METHOD PRIVATE ActionRun
VAR_INPUT
	tempActStep:ITFActStep;
END_VAR
VAR
END_VAR
VAR_STAT//此处定义静态变量, 保证每次进入该函数时能够在线监控当前值
	tempStep:DINT;
END_VAR
tempStep:=tempActStep.getStep();
CASE tempStep OF
0:
	IF tempActStep.isEx() THEN
		tempActStep.setBusyFlag();
		tempActStep.toBeginStep();
	END_IF
	t1(IN:= FALSE );
	t2(IN:= FALSE );
	t3(IN:= FALSE );
10:
	gShowLogTextTitle:='Chamber LL Vent';
	IF gRunningState<>RunningStatus.eErrorState THEN
		tempActStep.addStep(10,FALSE);
	ELSE
		gRunningLog.append(CONCAT('Chamber Vent POU Run:',DINT_TO_STRING(tempStep)));
		gRunningLog.append('Chamber Vent POU Run: Running State Error');
		error_Trigger(105);
		tempActStep.toDoneStep();
	END_IF
20:
	IF NOT gICP.ForeLineGauge.error AND gICP.ForeLineGauge.outputValue<gRoughtPumVaccum*10 THEN
		tempActStep.addStep(10,FALSE);
	ELSE
		error_Trigger(107);
		tempActStep.toDoneStep();
	END_IF
30:
	tempActStep.toStep(100,FALSE);
	gRoughRemain:=FALSE;
100:
	tempActStep.addStep(10,TRUE);
110:
	S_RoughPumping.Act_Init_Status();
	S_RoughPumping.Act_Ex();
	tempActStep.addStep(10,FALSE);
120:
	IF S_RoughPumping.done THEN
		tempActStep.addStep(2,FALSE);
	END_IF
	IF S_RoughPumping.errDone THEN
		tempActStep.toErrDoneStep();
	END_IF
122:
	tempActStep.addStep(2,TRUE);
124:
	IF gICP.TruboPum.Act_Close() THEN
		gRunningLog.append(CONCAT('Chamber Vent POU Run:',DINT_TO_STRING(tempStep)));
		gRunningLog.append('Chamber Vent POU Run: TruboPum Close');
		tempActStep.addStep(2,FALSE);
	END_IF
126:
	IF (gICP.TruboPum.Get_Done_Close() AND gICP.TruboPumNoRotation) AND 
		(NOT gICP.TruboPumAcc AND NOT gICP.TruboPumDcc AND NOT gICP.TruboPumNormal AND gICP.TruboPumNoRotation) THEN
		gRunningLog.append(CONCAT('Chamber Vent POU Run:',DINT_TO_STRING(tempStep)));
		gRunningLog.append('Chamber Vent POU Run: TruboPum Close Done');
		tempActStep.addStep(2,FALSE);
	END_IF
128:
	tempActStep.addStep(2,FALSE);
130:
	tempActStep.addStep(10,TRUE);
140:
	IF gICP.GateDoorValve.Get_Done_Ret() AND gICP.GateDoorRetSensor AND
		gICP.VentValve.Get_Done_Ret() AND NOT gICP.VentExtRelay AND
		gICP.SlowPummingValve.Get_Done_Ret() AND NOT gICP.SlowPummingExtRelay AND
		gICP.FastPummingValve.Get_Done_Ret() AND NOT gICP.FastPummingExtRelay AND
		gICP.ForlinLineValve.Get_Done_Ext() AND gICP.ForlinLineValveExtRelay AND////////////////
		gICP.RoughValve.Get_Done_Ret() AND NOT gICP.RoughValveExtRelay AND
		(gICP.PDV.Get_Done_Ext() OR gICP.PDVOpenSensor) AND gICP.PDVOpenSensor  THEN///////////////
		gRunningLog.append(CONCAT('Chamber Vent POU Run:',DINT_TO_STRING(tempStep)));
		gRunningLog.append('Chamber Vent POU Run: All Main Actuator Recovery');
		tempActStep.addStep(5,FALSE);		
	END_IF
145:
	IF gICP.PDV.Act_Retract() THEN
		gRunningLog.append(CONCAT('Chamber Vent POU Run:',DINT_TO_STRING(tempStep)));
		gRunningLog.append('Chamber Vent POU Run: PDV Close');
		tempActStep.addStep(2,FALSE);	
	END_IF
147:
	IF (gICP.PDV.Get_Done_Ret() OR gICP.PDVCloseSensor) THEN
		gRunningLog.append(CONCAT('Chamber Vent POU Run:',DINT_TO_STRING(tempStep)));
		gRunningLog.append('Chamber Vent POU Run: PDV Close DOne');
		tempActStep.addStep(3,FALSE);	
	END_IF
150:
	IF gICP.GateDoorValve.Act_Extend() THEN
		gRunningLog.append(CONCAT('Chamber Vent POU Run:',DINT_TO_STRING(tempStep)));
		gRunningLog.append('Chamber Vent POU Run: Gate Door Open');
		tempActStep.addStep(10,FALSE);	
	END_IF
160:
	IF gICP.GateDoorValve.Get_Done_Ext() AND gICP.GateDoorExtSensor THEN
		gRunningLog.append(CONCAT('Chamber Vent POU Run:',DINT_TO_STRING(tempStep)));
		gRunningLog.append('Chamber Vent POU Run: Gate Door Open Done');
		tempActStep.addStep(10,FALSE);	
	END_IF
170:
	tempActStep.addStep(10,TRUE);
180:
	tempActStep.toStep(220,FALSE);	
220:
	IF gICP.VentValve.Act_Extend() THEN
		gRunningLog.append(CONCAT('Chamber Vent POU Run:',DINT_TO_STRING(tempStep)));
		gRunningLog.append('Chamber Vent POU Run: Vent Valve Open');
		gRoughRemain:=FALSE;
		gRoughRemainTMPCanOpen:=FALSE;
		ups_CX51X0.Act_Wrtie();
		tempActStep.addStep(10,FALSE);
	END_IF
230:
	IF gICP.VentValve.Get_Done_Ext() THEN
		gRunningLog.append(CONCAT('Chamber Vent POU Run:',DINT_TO_STRING(tempStep)));
		gRunningLog.append('Chamber Vent POU Run: Vent Valve Open Done');
		tempActStep.addStep(10,FALSE);
	END_IF
240:
	t2(IN:= gICP.LoadLockGauge.outputValue>gATMPressure,PT:=T#120S );
	IF t2.Q OR NOT gICP.I_LLSwitch THEN
		t1(IN:= FALSE );
		t2(IN:= FALSE );
		t3(IN:= FALSE );
		gRunningLog.append(CONCAT('Chamber Vent POU Run:',DINT_TO_STRING(tempStep)));
		gRunningLog.append(CONCAT('Chamber Vent POU Run:LL Vent Pressure Arrive：',REAL_TO_STRING(gICP.LoadLockGauge.outputValue)));
		tempActStep.addStep(10,FALSE);
		RETURN;
	END_IF
	t1(IN:= TRUE,PT:=timeOutTime );
	IF t1.Q THEN
		t1(IN:= FALSE );
		t2(IN:= FALSE );
		t3(IN:= FALSE );
		error_Trigger(108);
//		tempActStep.toStep(170,FALSE);
		tempActStep.toDoneStep();
		RETURN;
	END_IF
250:
	tempActStep.addStep(10,TRUE);
260:
	IF gICP.VentValve.Act_Retract() THEN
		gRunningLog.append(CONCAT('Chamber Vent POU Run:',DINT_TO_STRING(tempStep)));
		gRunningLog.append('Chamber Vent POU Run: Vent Valve Close');
		tempActStep.addStep(10,FALSE);
	END_IF
270:
	IF gICP.VentValve.Get_Done_Ret() THEN
		gRunningLog.append(CONCAT('Chamber Vent POU Run:',DINT_TO_STRING(tempStep)));
		gRunningLog.append('Chamber Vent POU Run: Vent Valve Close Done');
		tempActStep.addStep(10,FALSE);
	END_IF
280:
	t3(IN:=TRUE,PT:=T#1S);
	IF t3.Q THEN
		t1(IN:= FALSE );
		t2(IN:= FALSE );
		t3(IN:= FALSE );
		tempActStep.addStep(10,FALSE);
	END_IF
290:
	tempActStep.addStep(10,TRUE);
300:
	IF gICP.GateDoorValve.Act_Retract() THEN
		gRunningLog.append(CONCAT('Chamber Vent POU Run:',DINT_TO_STRING(tempStep)));
		gRunningLog.append('Chamber Vent POU Run: Gate Door Close');
		tempActStep.addStep(10,FALSE);
	END_IF
310:
	IF gICP.GateDoorValve.Get_Done_Ret() THEN
		gRunningLog.append(CONCAT('Chamber Vent POU Run:',DINT_TO_STRING(tempStep)));
		gRunningLog.append('Chamber Vent POU Run: Gate Door Close Done');
		tempActStep.addStep(10,FALSE);
	END_IF
320:
	tempActStep.toStep(370,FALSE);
370:
	tempActStep.addStep(10,TRUE);
380:
	IF gICP.ForlinLineValve.Act_Extend() THEN
		gRunningLog.append(CONCAT('Chamber Vent POU Run:',DINT_TO_STRING(tempStep)));
		gRunningLog.append('Chamber Vent POU Run: ForLine Valve Open');
		tempActStep.addStep(10,FALSE);
	END_IF
390:
	IF gICP.ForlinLineValve.Get_Done_Ext() THEN
		gRunningLog.append(CONCAT('Chamber Vent POU Run:',DINT_TO_STRING(tempStep)));
		gRunningLog.append('Chamber Vent POU Run: ForLine Valve Open Done');
		tempActStep.addStep(10,FALSE);
	END_IF
400:
	tempActStep.toStep(1000,FALSE);
1000:
	tempActStep.toDoneStep();

60000://Done
	tempActStep.setDoneFlag();
	tempActStep.toZeroStep();
	
65000://Error
	tempActStep.setErrDoneFlag();
	tempActStep.toZeroStep();
	gICP.VentValve.Act_Retract();
END_CASE
END_METHOD

END_PROGRAM

// ---- POUs/MachinePOU/SemiAutomatic/S_MachineVent.TcPOU
PROGRAM S_MachineVent
VAR_INPUT
	bInit				:BOOL:=FALSE;// 初始化状态 busy/done/errDone
	bTrig				:BOOL:=FALSE;// 执行触发 信号
	bReset				:BOOL:=FALSE;// 报错 复位
	bPause				:BOOL:=FALSE;// 暂停 运行
	bStop				:BOOL:=FALSE;// 停止 运行
	bAbort				:BOOL:=FALSE;// 中止 运行
	
END_VAR
VAR_OUTPUT
	busy				:BOOL;
	done				:BOOL;
	errDone				:BOOL;
END_VAR
VAR
	actStep				:ActStepBase;
END_VAR
VAR
	i: INT;
	t1:ton;
	t2:ton;
	t3:ton;
	notchoose:BOOL;
	timeOutTime:TIME:=T#120S;
	safecheckTime:TIME:=T#1S;
END_VAR

busy:=actStep.isBusy();
done:=actStep.isDone();
errDone:=actStep.isError();
actStep.Act_Pause(pause:=bPause);

IF bTrig THEN
	bTrig:=FALSE;
	IF NOT busy THEN
		actStep.Act_ex();
	END_IF
END_IF

//状态复位
IF bInit THEN
	bInit:=FALSE;
	Act_init_status();
END_IF

IF bAbort OR bStop THEN
	bAbort:=FALSE;
	bStop:=FALSE;
	Act_init_status();
	actStep.toZeroStep();
	gShowLogTextTitle:='NON';
END_IF
ActionRun(tempActStep:=actStep);

(*
---Trigger action
*)
METHOD Act_Ex : BOOL
VAR_INPUT
END_VAR
IF NOT busy THEN
	actStep.Act_ex();
	Act_Ex:=TRUE;
ELSE
	Act_Ex:=FALSE;
END_IF
END_METHOD

(*
---功能: 状态复位 busy/done/errDone;
*)
METHOD Act_Init_Status
VAR_INPUT
END_VAR
actStep.Act_Init();
END_METHOD

METHOD PRIVATE ActionRun
VAR_INPUT
	tempActStep:ITFActStep;
END_VAR
VAR
END_VAR
VAR_STAT//此处定义静态变量, 保证每次进入该函数时能够在线监控当前值
	tempStep:DINT;
END_VAR
tempStep:=tempActStep.getStep();
CASE tempStep OF
0:
	IF tempActStep.isEx() THEN
		tempActStep.setBusyFlag();
		tempActStep.toBeginStep();
	END_IF
	t1(IN:= FALSE );
	t2(IN:= FALSE );
	t3(IN:= FALSE );
10:
	gShowLogTextTitle:='Machine Vent';
	IF gRunningState<>RunningStatus.eErrorState THEN
		tempActStep.addStep(10,FALSE);
	ELSE
		error_Trigger(105);
		tempActStep.toErrDoneStep();
	END_IF
20:
	IF NOT gICP.ForeLineGauge.error AND gICP.ForeLineGauge.outputValue<gRoughtPumVaccum*10 THEN
		tempActStep.addStep(10,FALSE);
	ELSE
		error_Trigger(107);
		tempActStep.toErrDoneStep();
	END_IF
30:
	gRoughRemain:=FALSE;
	tempActStep.toStep(100,FALSE);
100:
	tempActStep.addStep(10,TRUE);
110:
	S_RoughPumping.Act_Init_Status();
	S_RoughPumping.Act_Ex();
	tempActStep.addStep(10,FALSE);
120:
	IF S_RoughPumping.done THEN
		gShowLogTextTitle:='Machine Vent';
		tempActStep.addStep(10,FALSE);
	END_IF
	IF S_RoughPumping.errDone THEN
		tempActStep.toErrDoneStep();
	END_IF
130:
	tempActStep.addStep(10,TRUE);
140:
	IF gICP.TruboPum.Act_Close() THEN
		gRunningLog.append(CONCAT('Machine Vent POU Run:',DINT_TO_STRING(tempStep)));
		gRunningLog.append('Machine Vent POU Run:TB Close');
		tempActStep.addStep(10,FALSE);
	END_IF
150:
	IF (gICP.TruboPum.Get_Done_Close() AND gICP.TruboPumNoRotation) AND (NOT gICP.TruboPumAcc AND NOT gICP.TruboPumDcc AND NOT gICP.TruboPumNormal AND gICP.TruboPumNoRotation) THEN
		gRunningLog.append(CONCAT('Machine Vent POU Run:',DINT_TO_STRING(tempStep)));
		gRunningLog.append('Machine Vent POU Run:TB Close Done');
		tempActStep.addStep(10,FALSE);
	END_IF
160:
	IF gICP.GateDoorValve.Get_Done_Ret() AND gICP.GateDoorRetSensor AND
		gICP.VentValve.Get_Done_Ret() AND NOT gICP.VentExtRelay AND
		gICP.SlowPummingValve.Get_Done_Ret() AND NOT gICP.SlowPummingExtRelay AND
		gICP.FastPummingValve.Get_Done_Ret() AND NOT gICP.FastPummingExtRelay AND
		gICP.ForlinLineValve.Get_Done_Ext() AND gICP.ForlinLineValveExtRelay AND
		gICP.RoughValve.Get_Done_Ret() AND NOT gICP.RoughValveExtRelay AND
		(gICP.PDV.Get_Done_Ext() OR gICP.PDVOpenSensor)  THEN
		gRunningLog.append(CONCAT('Machine Vent POU Run:',DINT_TO_STRING(tempStep)));
		gRunningLog.append('Machine Vent POU Run:Main Actuator Recovery');
		tempActStep.addStep(10,FALSE);		
	END_IF
170:
	IF gICP.GateDoorValve.Act_Extend() THEN
		gRunningLog.append(CONCAT('Machine Vent POU Run:',DINT_TO_STRING(tempStep)));
		gRunningLog.append('Machine Vent POU Run:Gate Door Open');
		tempActStep.addStep(10,FALSE);	
	END_IF
180:
	IF gICP.GateDoorValve.Get_Done_Ext() AND gICP.GateDoorExtSensor THEN
		gRunningLog.append(CONCAT('Machine Vent POU Run:',DINT_TO_STRING(tempStep)));
		gRunningLog.append('Machine Vent POU Run:Gate Door Open Done');
		tempActStep.addStep(10,FALSE);	
	END_IF
190:
	tempActStep.addStep(10,TRUE);
200:
	tempActStep.addStep(10,FALSE);
210:
	IF gICP.PDV.Act_Open() THEN
		gRunningLog.append(CONCAT('Machine Vent POU Run:',DINT_TO_STRING(tempStep)));
		gRunningLog.append('Machine Vent POU Run:PDV Open');
		tempActStep.addStep(2,FALSE);
	END_IF
212:
	IF (gICP.PDV.Get_Done_Ext() OR gICP.PDVOpenSensor) THEN
		gRunningLog.append(CONCAT('Machine Vent POU Run:',DINT_TO_STRING(tempStep)));
		gRunningLog.append('Machine Vent POU Run:PDV Open Done');
		tempActStep.addStep(2,FALSE);
	END_IF
214:
	tempActStep.addStep(2,TRUE);
216:
	IF gICP.ForlinLineValve.Act_Retract() THEN
		gRunningLog.append(CONCAT('Machine Vent POU Run:',DINT_TO_STRING(tempStep)));
		gRunningLog.append('Machine Vent POU Run:ForeLine Valve Close');
		tempActStep.addStep(2,FALSE);
	END_IF
218:
	IF gICP.ForlinLineValve.Get_Done_Ret() THEN
		gRunningLog.append(CONCAT('Machine Vent POU Run:',DINT_TO_STRING(tempStep)));
		gRunningLog.append('Machine Vent POU Run:ForeLine Valve Close Done');
		tempActStep.addStep(2,FALSE);
	END_IF
220:
	IF gICP.VentValve.Act_Extend() THEN
		gRunningLog.append(CONCAT('Machine Vent POU Run:',DINT_TO_STRING(tempStep)));
		gRunningLog.append('Machine Vent POU Run:Vent Valve Open');
		gRoughRemain:=FALSE;
		gRoughRemainTMPCanOpen:=FALSE;
		ups_CX51X0.Act_Wrtie();
		tempActStep.addStep(10,FALSE);
	END_IF
230:
	IF gICP.VentValve.Get_Done_Ext() THEN
		gRunningLog.append(CONCAT('Machine Vent POU Run:',DINT_TO_STRING(tempStep)));
		gRunningLog.append('Machine Vent POU Run:Vent Valve Open Done');
		tempActStep.addStep(10,FALSE);
	END_IF
240:
	t2(IN:= gICP.LoadLockGauge.outputValue>gATMPressure,PT:=T#180S );
	IF t2.Q OR NOT gICP.I_LLSwitch THEN
		t1(IN:= FALSE );
		t2(IN:= FALSE );
		t3(IN:= FALSE );
		gRunningLog.append(CONCAT('Machine Vent POU Run:',DINT_TO_STRING(tempStep)));
		gRunningLog.append(CONCAT('Machine Vent POU Run:LL Vent Pressure Arrive：',REAL_TO_STRING(gICP.LoadLockGauge.outputValue)));
		tempActStep.addStep(10,FALSE);
		RETURN;
	END_IF
	t1(IN:= TRUE,PT:=timeOutTime );
	IF t1.Q THEN
		t1(IN:= FALSE );
		t2(IN:= FALSE );
		t3(IN:= FALSE );
		error_Trigger(112);
//		tempActStep.toStep(214,FALSE);
		tempActStep.toDoneStep();
		RETURN;
	END_IF
250:
	tempActStep.addStep(10,TRUE);
260:
	IF gICP.VentValve.Act_Retract() THEN
		gRunningLog.append(CONCAT('Machine Vent POU Run:',DINT_TO_STRING(tempStep)));
		gRunningLog.append('Machine Vent POU Run:Vent Valve Close');
		tempActStep.addStep(10,FALSE);
	END_IF
270:
	IF gICP.VentValve.Get_Done_Ret() THEN
		gRunningLog.append(CONCAT('Machine Vent POU Run:',DINT_TO_STRING(tempStep)));
		gRunningLog.append('Machine Vent POU Run:Vent Valve Close Done');
		tempActStep.addStep(10,FALSE);
	END_IF
280:
	t3(IN:=TRUE,PT:=T#1S);
	IF t3.Q THEN
		t1(IN:= FALSE );
		t2(IN:= FALSE );
		t3(IN:= FALSE );
		tempActStep.addStep(10,FALSE);
	END_IF
290:
	tempActStep.addStep(10,TRUE);
300:
	IF gICP.GateDoorValve.Act_Retract() THEN
		gRunningLog.append(CONCAT('Machine Vent POU Run:',DINT_TO_STRING(tempStep)));
		gRunningLog.append('Machine Vent POU Run:Gate Door Close');
		tempActStep.addStep(10,FALSE);
	END_IF
310:
	IF gICP.GateDoorValve.Get_Done_Ret() THEN
		gRunningLog.append(CONCAT('Machine Vent POU Run:',DINT_TO_STRING(tempStep)));
		gRunningLog.append('Machine Vent POU Run:Gate Door Close Done');
		tempActStep.addStep(10,FALSE);
	END_IF
320:
	tempActStep.toStep(370,FALSE);
370:
	tempActStep.addStep(10,TRUE);
380:
	IF gICP.PDV.Act_Retract() THEN
		gRunningLog.append(CONCAT('Machine Vent POU Run:',DINT_TO_STRING(tempStep)));
		gRunningLog.append('Machine Vent POU Run:PDV Close');
		tempActStep.addStep(10,FALSE);
	END_IF
390:
	IF (gICP.PDV.Get_Done_Ret() OR gICP.PDVCloseSensor) THEN
		gRunningLog.append(CONCAT('Machine Vent POU Run:',DINT_TO_STRING(tempStep)));
		gRunningLog.append('Machine Vent POU Run:PDV Close Done');
		tempActStep.addStep(10,FALSE);
	END_IF
400:
	tempActStep.toStep(1000,FALSE);
1000:
	tempActStep.toDoneStep();

60000://Done
	tempActStep.setDoneFlag();
	tempActStep.toZeroStep();
	
65000://Error
	tempActStep.setErrDoneFlag();
	tempActStep.toZeroStep();
	gICP.VentValve.Act_Retract();
END_CASE
END_METHOD

END_PROGRAM

// ---- POUs/MachinePOU/SemiAutomatic/S_Etching.TcPOU
PROGRAM S_Etching
VAR_INPUT
	bInit				:BOOL:=FALSE;// 初始化状态 busy/done/errDone
	bTrig				:BOOL:=FALSE;// 执行触发 信号
	bReset				:BOOL:=FALSE;// 报错 复位
	bPause				:BOOL:=FALSE;// 暂停 运行
	bStop				:BOOL:=FALSE;// 停止 运行
	bAbort				:BOOL:=FALSE;// 中止 运行
	
END_VAR
VAR_OUTPUT
	busy				:BOOL;
	done				:BOOL;
	errDone				:BOOL;
END_VAR
VAR
	actStep				:ActStepBase;
END_VAR
VAR
	i: INT;
	t1:ton;
	t2:ton;
	t3:ton;
	notchoose:BOOL;
	timeOutTime:TIME:= T#120S;
	ventTime:TIME:=T#15S;
	safecheckTime:TIME:=T#2S;
	currentTimes:INT:=1;
	rfComControl:TON;
	rTrig:R_TRIG;
END_VAR

busy:=actStep.isBusy();
done:=actStep.isDone();
errDone:=actStep.isError();
actStep.Act_Pause(pause:=bPause);

IF bTrig THEN
	bTrig:=FALSE;
	IF NOT busy THEN
		actStep.Act_ex();
	END_IF
END_IF

//状态复位
IF bInit THEN
	bInit:=FALSE;
	Act_init_status();
END_IF

IF bAbort OR bStop THEN
	bAbort:=FALSE;
	bStop:=FALSE;
	Act_init_status();
	actStep.toZeroStep();
	S_CO_ControlRF.bStop:=TRUE;
	S_CO_ControlRF.bAbort:=TRUE;
	gRFComControl:=FALSE;
	gShowLogTextTitle:='NON';
END_IF
ActionRun(tempActStep:=actStep);
IF gRFComControl AND gICP.SourceRF.openRelay AND gICP.powerRF.openRelay THEN
	rfComControl(IN:=gICP.SourceRF.Get_Done_Open() AND gICP.PowerRF.Get_Done_Open(),PT:=UDINT_TO_TIME(gRFSetTime*1000));// 反射调整超时时间
	gRFRemainTime:=TIME_TO_UDINT(rfComControl.ET/1000);
	gRFRemainTime:=gRFSetTime-gRFRemainTime;
END_IF
rTrig(CLK:=gRFRemainTime=0);
IF rTrig.Q THEN
	gICP.SourceRF.Act_Close();
	gICP.PowerRF.Act_Close();
	gRFComControl:=FALSE;
END_IF

(*
---Trigger action
*)
METHOD Act_Ex : BOOL
VAR_INPUT
END_VAR
IF NOT busy THEN
	actStep.Act_ex();
	Act_Ex:=TRUE;
ELSE
	Act_Ex:=FALSE;
END_IF
END_METHOD

(*
---功能: 状态复位 busy/done/errDone;
*)
METHOD Act_Init_Status
VAR_INPUT
END_VAR
actStep.Act_Init();
END_METHOD

METHOD PRIVATE ActionRun
VAR_INPUT
	tempActStep:ITFActStep;
END_VAR
VAR_STAT//此处定义静态变量, 保证每次进入该函数时能够在线监控当前值
	tempStep:DINT;
END_VAR
tempStep:=tempActStep.getStep();
CASE tempStep OF
0:
	IF tempActStep.isEx() THEN
		tempActStep.setBusyFlag();
		tempActStep.toBeginStep();
	END_IF
	currentTimes:=1;
	t1(IN:= FALSE );
	t2(IN:= FALSE );
	t3(IN:= FALSE );
10:
	gShowLogTextTitle:='Etching';
	IF gRunningState<>RunningStatus.eErrorState THEN
		tempActStep.addStep(10,FALSE);
	ELSE
		error_Trigger(105);
	END_IF
	currentTimes:=1;
20:
	IF ControlMode.eSemiAutoMode=gCtrlMode OR ControlMode.eManualCtrMode=gCtrlMode THEN
		S_RoughPumping.Act_Init_Status();
		S_RoughPumping.Act_Ex();
		tempActStep.addStep(10,FALSE);
	ELSIF( ControlMode.eAutoCtrMode=gCtrlMode) THEN
		S_RoughPumping.Act_Init_Status();
		S_RoughPumping.Act_Ex();
		tempActStep.addStep(10,FALSE);
	ELSE
		tempActStep.toErrDoneStep();
	END_IF
30:
	IF S_RoughPumping.done THEN
		gShowLogTextTitle:='Etching';
		tempActStep.addStep(5,FALSE);
	END_IF
	IF S_RoughPumping.errDone THEN
		tempActStep.toErrDoneStep();
	END_IF	
35:
	tempActStep.addStep(5,TRUE);
40:
	IF gICP.HeMFC_SetFlowHMI<1 THEN
		tempActStep.toErrDoneStep();
		error_Trigger(200);
	ELSE
		tempActStep.addStep(10,FALSE);
	END_IF
50:// 记忆状态判断
	IF gWaferMemoryState=2 THEN
		gRunningLog.append(CONCAT('Etching POU Run:',DINT_TO_STRING(tempStep)));
		gRunningLog.append('Etching POU Run: wafer in chamber and etch done');
		tempActStep.toDoneStep();
	ELSIF gWaferMemoryState=1 THEN
		gRunningLog.append(CONCAT('Etching POU Run:',DINT_TO_STRING(tempStep)));
		gRunningLog.append('Etching POU Run: Wafer in chamber and no etch ');
		tempActStep.toStep(100,FALSE);// 直接进行Etch
	ELSIF gWaferMemoryState=0 THEN	
//		tempActStep.addStep(10,FALSE);// 先进行Load
		error_Trigger(116);
		tempActStep.toErrDoneStep();
	END_IF
100:
	tempActStep.addStep(10,TRUE);
110:
	tempActStep.addStep(10,FALSE);
120:
	IF NOT gICP.ForeLineGauge.error AND NOT gICP.LoadLockGauge.error AND NOT gICP.AIMGauge.error THEN
		tempActStep.addStep(10,FALSE);
	ELSE
		error_Trigger(107);
		tempActStep.toStep(10,FALSE);
	END_IF
130:
	IF gICP.ForlinLineValve.Act_Extend() AND gICP.PDV.Act_Open() THEN
		gRunningLog.append(CONCAT('Etching POU Run:',DINT_TO_STRING(tempStep)));
		gRunningLog.append('Etching POU Run: ForeLine Valve and PDV Open');
		tempActStep.addStep(10,FALSE);
	END_IF
140:
	IF (gICP.PDV.Get_Done_Ext() OR gICP.PDVOpenSensor) AND gICP.PDVOpenRelay AND gICP.ForlinLineValve.Get_Done_Ext() THEN
		gRunningLog.append(CONCAT('Etching POU Run:',DINT_TO_STRING(tempStep)));
		gRunningLog.append('Etching POU Run: ForeLine Valve and PDV Open Done');
		tempActStep.addStep(10,FALSE);
	END_IF
150:
	tempActStep.toStep(230,FALSE);	
230:
	tempActStep.addStep(10,TRUE);
240:	
	IF gICP.TruboPumNoRotation OR NOT(gICP.TruboPumAcc OR gICP.TruboPumDcc OR gICP.TruboPumNormal) AND FALSE THEN  //  临时屏蔽用
		IF gICP.TruboPum.Act_Open() THEN
			tempActStep.addStep(10,FALSE);
			gRunningLog.append(CONCAT('Etching POU Run:',DINT_TO_STRING(tempStep)));
			gRunningLog.append('Etching POU Run: TruboPum is not open');
		END_IF
	ELSE
		tempActStep.toStep(260,FALSE);
	END_IF
250:
	IF gICP.TruboPum.Get_Done_Open() AND gICP.TruboPumNormal AND gICP.TruboPumRotationSpeed>440 THEN
		gRunningLog.append(CONCAT('Etching POU Run:',DINT_TO_STRING(tempStep)));
		gRunningLog.append('Etching POU Run: TruboPum open Done');
		tempActStep.addStep(10,FALSE);
	END_IF
	IF  gICP.TruboPum.error THEN
		tempActStep.toErrDoneStep();
	END_IF
260:
	tempActStep.addStep(30,TRUE);//  临时屏蔽用
270:
	IF gICP.AIMValve.Act_Extend() THEN
		gRunningLog.append(CONCAT('Etching POU Run:',DINT_TO_STRING(tempStep)));
		gRunningLog.append('Etching POU Run:AIM Gauge open');
		tempActStep.addStep(10,FALSE);
	END_IF
280:
	t2(IN:= gICP.AIMGauge.outputValue<gUltimateVacuum AND gICP.AIMValve.Get_Done_Ext(),PT:=safecheckTime );
	IF t2.Q THEN
		t1(IN:= FALSE );
		t2(IN:= FALSE );
		t3(IN:= FALSE );
		gRunningLog.append(CONCAT('Etching POU Run:',DINT_TO_STRING(tempStep)));
		gRunningLog.append('Etching POU Run:AIM Gauge open Done and Preessure is Arrive');
		tempActStep.addStep(10,FALSE);
		RETURN;
	END_IF
	t3(IN:= TRUE,PT:=timeOutTime );
	IF t3.Q THEN
		t1(IN:= FALSE );
		t2(IN:= FALSE );
		t3(IN:= FALSE );
		error_Trigger(123);
		tempActStep.toErrDoneStep();
		RETURN;
	END_IF	
290:
	tempActStep.addStep(10,TRUE);
300:
	IF gICP.AIMValve.Act_Retract() THEN
		gRunningLog.append(CONCAT('Etching POU Run:',DINT_TO_STRING(tempStep)));
		gRunningLog.append('Etching POU Run:AIM Gauge Close');
		tempActStep.addStep(10,FALSE);
	END_IF
310:
	IF gICP.AIMValve.Get_Done_Ret() THEN
		gRunningLog.append(CONCAT('Etching POU Run:',DINT_TO_STRING(tempStep)));
		gRunningLog.append('Etching POU Run:AIM Gauge Close Done');
		tempActStep.addStep(10,FALSE);
	END_IF
320:
	tempActStep.addStep(10,TRUE);
330:
	IF gICP.LiftPinCyl.Act_Retract() THEN
		gRunningLog.append(CONCAT('Etching POU Run:',DINT_TO_STRING(tempStep)));
		gRunningLog.append('Etching POU Run:Lift PIN Down');
		tempActStep.addStep(10,FALSE);
	END_IF
340:
	IF gICP.LiftPinCyl.Get_Done_Ret() THEN
		tempActStep.addStep(10,FALSE);
	END_IF
350:
	tempActStep.addStep(10,TRUE);
360:
	IF gICP.ElectrodeCyl.Act_Extend() THEN
		gRunningLog.append(CONCAT('Etching POU Run:',DINT_TO_STRING(tempStep)));
		gRunningLog.append('Etching POU Run:ElectrodeCyl Up');
		tempActStep.addStep(10,FALSE);
	END_IF
370:
	IF gICP.ElectrodeCyl.Get_Done_Ext() THEN
		tempActStep.addStep(2,FALSE);
	END_IF
372:
	tempActStep.addStep(2,TRUE);
374:
	IF gICP.HeINValve.Act_Extend() THEN
		tempActStep.addStep(2,FALSE);
	END_IF
376:
	IF gICP.HeINValve.Get_Done_Ext() THEN
		tempActStep.addStep(2,FALSE);
	END_IF
378:
	tempActStep.addStep(2,FALSE);
380:
	tempActStep.addStep(10,TRUE);
390:
	IF currentTimes<=gShowNum THEN
		gICP.MFC1.setFlow:=STRING_TO_UDINT(gRecipeViewData[currentTimes].mfc1);
		gICP.MFC2.setFlow:=STRING_TO_UDINT(gRecipeViewData[currentTimes].mfc2);
		gICP.MFC3.setFlow:=STRING_TO_UDINT(gRecipeViewData[currentTimes].mfc3);
		gICP.MFC4.setFlow:=STRING_TO_UDINT(gRecipeViewData[currentTimes].mfc4);
		gICP.MFC5.setFlow:=STRING_TO_UDINT(gRecipeViewData[currentTimes].mfc5);
		gICP.MFC6.setFlow:=STRING_TO_UDINT(gRecipeViewData[currentTimes].mfc6);
		gICP.MFC7.setFlow:=STRING_TO_UDINT(gRecipeViewData[currentTimes].mfc7);
		gICP.MFC8.setFlow:=STRING_TO_UDINT(gRecipeViewData[currentTimes].mfc8);
		gICP.MFC9.setFlow:=STRING_TO_UDINT(gRecipeViewData[currentTimes].mfc9);
		tempActStep.addStep(10,FALSE);
		gRunningLog.append(CONCAT('Etching POU Run:',DINT_TO_STRING(tempStep)));
		gRunningLog.append('Etching POU Run:Set MFC Par');
		gRunningLog.append(CONCAT('Etching POU Run:',DINT_TO_STRING(tempStep)));
		gRunningLog.append(CONCAT('Etching POU Run:Current step is  ',INT_TO_STRING(currentTimes)));
	ELSE
		tempActStep.toStep(800,FALSE);////////////////////////////////////////////Done
	END_IF
	
400:
	IF gICP.S_GASBOX_AllMFCClearDoneStep THEN
		gICP.C_GASBOX_AllMFCSet:=TRUE;
		gICP.S_GASBOX_AllMFCSetDone:=FALSE;
		tempActStep.addStep(10,FALSE);
	END_IF
410:
	IF NOT gICP.C_GASBOX_AllMFCSet THEN
		tempActStep.addStep(10,FALSE);
	END_IF
420:
	IF gICP.S_GASBOX_AllMFCSetDone THEN
		gRunningLog.append(CONCAT('Etching POU Run:',DINT_TO_STRING(tempStep)));
		gRunningLog.append('Etching POU Run:Set MFC Par Done');
		tempActStep.addStep(10,FALSE);
	END_IF
430:
	tempActStep.addStep(10,TRUE);
440:
	gICP.C_GASBOX_AllGVAOpen:=TRUE;
	gRunningLog.append(CONCAT('Etching POU Run:',DINT_TO_STRING(tempStep)));
	gRunningLog.append('Etching POU Run:GAS Box GVA Open');
	tempActStep.addStep(10,FALSE);
450:
	IF gICP.S_GASBOX_AllGVAOpen THEN
		gRunningLog.append(CONCAT('Etching POU Run:',DINT_TO_STRING(tempStep)));
		gRunningLog.append('Etching POU Run:GAS Box GVA Open Done');
		tempActStep.addStep(10,FALSE);
	END_IF
460:
	t1(IN:=TRUE ,PT:=T#4S);
	IF t1.Q THEN
		t1(IN:= FALSE );
		t2(IN:= FALSE );
		t3(IN:= FALSE );
		tempActStep.addStep(10,FALSE);
	END_IF
470:
	IF gICP.S_GASBOX_AllMFCClearDone THEN// 全部MFC实际流量小于1
		tempActStep.addStep(10,FALSE);
		gRunningLog.append(CONCAT('Etching POU Run:',DINT_TO_STRING(tempStep)));
		gRunningLog.append('Etching POU Run:GAS Box GVB MFC flow is clear done');
	END_IF
480:
	tempActStep.addStep(10,TRUE);
490:
	gICP.C_GASBOX_AllGVBOpen:=TRUE;
	gRunningLog.append(CONCAT('Etching POU Run:',DINT_TO_STRING(tempStep)));
	gRunningLog.append('Etching POU Run:GAS Box GVB Open');
	tempActStep.addStep(10,FALSE);
500:
	IF gICP.S_GASBOX_AllGVBOpen THEN
		gRunningLog.append(CONCAT('Etching POU Run:',DINT_TO_STRING(tempStep)));
		gRunningLog.append('Etching POU Run:GAS Box GVB Open Done');
		tempActStep.addStep(10,FALSE);
	END_IF
510:	
	t1(IN:=TRUE ,PT:=T#4S);
	IF t1.Q THEN
		t1(IN:= FALSE );
		t2(IN:= FALSE );
		t3(IN:= FALSE );
		tempActStep.addStep(10,FALSE);
	END_IF
520:
	IF gICP.S_GASBOX_AllMFCSetEqual THEN
		gRunningLog.append(CONCAT('Etching POU Run:',DINT_TO_STRING(tempStep)));
		gRunningLog.append('Etching POU Run:GAS Box MFC Set Flow is arrive');
		tempActStep.addStep(10,FALSE);
	END_IF
530:
	tempActStep.addStep(10,TRUE);
540:
	IF gICP.ISOValve.Act_Extend() THEN
		gRunningLog.append(CONCAT('Etching POU Run:',DINT_TO_STRING(tempStep)));
		gRunningLog.append('Etching POU Run:ISO Valve Open');
		tempActStep.addStep(10,FALSE);
	END_IF
550:
	IF gICP.ISOValve.Get_Done_Ext() THEN
		tempActStep.addStep(10,FALSE);
	END_IF
560:
	tempActStep.addStep(10,TRUE);
570:
	gICP.PDV.Act_ChangePre(STRING_TO_REAL(gRecipeViewData[currentTimes].pdvPoint));
	gRunningLog.append(CONCAT('Etching POU Run:',DINT_TO_STRING(tempStep)));
	gRunningLog.append('Etching POU Run:PDV is change mode to preessur mode');
	tempActStep.addStep(10,FALSE);
580:
	IF gICP.PDV.Get_Done_Mode() THEN
		tempActStep.addStep(10,FALSE);
	END_IF
590:
	tempActStep.addStep(5,TRUE);
595:
	IF NOT gICP.S_MFCMonitFlowNotZero THEN
		tempActStep.addStep(5,FALSE);
	ELSE
		error_Trigger(120);
		tempActStep.toStep(590,FALSE);
		RETURN;
	END_IF
600:
	gRunningLog.append(CONCAT('Etching POU Run:',DINT_TO_STRING(tempStep)));
	gRunningLog.append('Etching POU Run:Set RF Par');
	gICP.SourceRF.HMIItf.setpower:=STRING_TO_UDINT(gRecipeViewData[currentTimes].rfPoint_Source);
	gICP.SourceRF.setpower:=gICP.SourceRF.HMIItf.setpower;
	gICP.SourceRF.Act_Write();
	tempActStep.addStep(10,FALSE);
610:
	IF gICP.SourceRF.HMIItf.setpower=gICP.SourceRF.setpower AND gICP.SourceRF.setpower=gICP.SourceRF.setpowerRead THEN
		tempActStep.addStep(10,FALSE);
	END_IF
620:
	gICP.PowerRF.HMIItf.setpower:=STRING_TO_UDINT(gRecipeViewData[currentTimes].rfPoint_Power);
	gICP.PowerRF.setpower:=gICP.PowerRF.HMIItf.setpower;
	gICP.PowerRF.Act_Write();
	gCO_ControlRFTime:=STRING_TO_UDINT(gRecipeViewData[currentTimes].etchTime);
	tempActStep.addStep(10,FALSE);
630:
	IF gICP.PowerRF.HMIItf.setpower=gICP.PowerRF.setpower AND gICP.PowerRF.setpower=gICP.PowerRF.setpowerRead THEN
		tempActStep.addStep(10,FALSE);
	END_IF
640:
	tempActStep.addStep(10,FALSE);
650:
	S_CO_ControlRF.Act_Init_Status();
	S_CO_ControlRF.Act_Ex();
	gRunningLog.append(CONCAT('Etching POU Run:',DINT_TO_STRING(tempStep)));
	gRunningLog.append('Etching POU Run:RF Open');
	tempActStep.addStep(5,FALSE);
655:
	IF S_CO_ControlRF.busy THEN
		tempActStep.addStep(5,FALSE);
	END_IF
660:
	IF S_CO_ControlRF.done THEN
		gRunningLog.append(CONCAT('Etching POU Run:',DINT_TO_STRING(tempStep)));
		gRunningLog.append('Etching POU Run:Etch Done');
		tempActStep.addStep(10,FALSE);
		RETURN;
	END_IF
	IF S_CO_ControlRF.errDone THEN
		gCO_ControlRFTimeRemain:=gCO_ControlRFTime;
		tempActStep.toStep(590,FALSE);
	END_IF	
665://  临时屏蔽用
	t1(IN:=TRUE ,PT:=T#10S);
	IF t1.Q THEN
		t1(IN:= FALSE );
		t2(IN:= FALSE );
		t3(IN:= FALSE );
		tempActStep.addStep(5,FALSE);
	END_IF
670:////////////////关气，关其他的东西，还原
	tempActStep.addStep(10,TRUE);
680:
	gICP.C_GASBOX_AllGVBClose:=TRUE;
	gRunningLog.append(CONCAT('Etching POU Run:',DINT_TO_STRING(tempStep)));
	gRunningLog.append('Etching POU Run:Gas Box GVB close');
	tempActStep.addStep(2,FALSE);
682:
	tempActStep.addStep(2,TRUE);
684:
	IF gICP.ForlinLineValve.Act_Extend() AND gICP.PDV.Act_Open() THEN
		gRunningLog.append(CONCAT('Etching POU Run:',DINT_TO_STRING(tempStep)));
		gRunningLog.append('Etching POU Run:PDV and ForeLine Open');
		tempActStep.addStep(2,FALSE);
	END_IF
686:
	IF gICP.ForlinLineValve.Get_Done_Ext() AND (gICP.PDV.Get_Done_Ext() OR gICP.PDVOpenSensor) THEN
//		gICP.PDV.Act_ChangePos();
		tempActStep.addStep(4,FALSE);
	END_IF
690:
	IF gICP.S_GASBOX_AllMFCClearDone THEN
		gRunningLog.append(CONCAT('Etching POU Run:',DINT_TO_STRING(tempStep)));
		gRunningLog.append('Etching POU Run:Gas Box flow is cleared done');
		tempActStep.addStep(10,FALSE);
	END_IF
700:
	t1(IN:=TRUE ,PT:=T#2S);
	IF t1.Q THEN
		t1(IN:= FALSE );
		t2(IN:= FALSE );
		t3(IN:= FALSE );
		tempActStep.addStep(10,FALSE);
	END_IF
710:
	tempActStep.addStep(10,TRUE);
720:
	gICP.C_GASBOX_AllMFCClear:=TRUE;
	gRunningLog.append(CONCAT('Etching POU Run:',DINT_TO_STRING(tempStep)));
	gRunningLog.append('Etching POU Run:Gas Box set flow is cleared');
	tempActStep.addStep(10,FALSE);
730:
	IF gICP.S_GASBOX_AllMFCClearDone THEN
		tempActStep.addStep(10,FALSE);
	END_IF
740:
	gICP.C_GASBOX_AllGVAClose:=TRUE;
	gRunningLog.append(CONCAT('Etching POU Run:',DINT_TO_STRING(tempStep)));
	gRunningLog.append('Etching POU Run:Gas Box GVA Close');
	tempActStep.addStep(10,FALSE);
750:
	t1(IN:=TRUE ,PT:=T#2S);
	IF t1.Q THEN
		t1(IN:= FALSE );
		t2(IN:= FALSE );
		t3(IN:= FALSE );
		tempActStep.addStep(10,FALSE);
	END_IF
760:
	tempActStep.addStep(10,TRUE);
770:
	tempActStep.addStep(10,FALSE);
780:
//	IF gICP.PDV.ReadState=XXX THEN // PDV 模式切换完成
//		tempActStep.addStep(10,FALSE);
//	END_IF
	tempActStep.addStep(10,FALSE);
790:
	tempActStep.toStep(380,FALSE);
	currentTimes:=currentTimes+1;
	gRunningLog.append(CONCAT('Etching POU Run:',DINT_TO_STRING(tempStep)));
	gRunningLog.append(CONCAT('The current number of steps plus 1 ',''));
800:
	tempActStep.addStep(5,FALSE);
805:
	tempActStep.addStep(2,TRUE);
807:
	IF gICP.HeINValve.Act_Retract() THEN
		tempActStep.addStep(3,FALSE);
	END_IF
810:
	IF gICP.HeINValve.Get_Done_Ret() THEN
		tempActStep.addStep(2,FALSE);
	END_IF
812:
	tempActStep.addStep(2,TRUE);
814:
	IF gICP.HePumValve.Act_Extend() THEN
		tempActStep.addStep(2,FALSE);
	END_IF
816:
	IF gICP.HePumValve.Get_Done_Ext() THEN
		tempActStep.addStep(1,FALSE);
	END_IF
817:
	t2(IN:=TRUE ,PT:=T#2S);
	IF t2.Q THEN
		t1(IN:= FALSE );
		t2(IN:= FALSE );
		t3(IN:= FALSE );
		tempActStep.addStep(1,FALSE);
	END_IF
818:
	t1(IN:=gICP.HeMFC_ActFlow<1 AND gICP.HeCheckGaugeReal<1 ,PT:=T#2S);
	IF t1.Q THEN
		t1(IN:= FALSE );
		t2(IN:= FALSE );
		t3(IN:= FALSE );
		gICP.HePumValve.Act_Retract();
		tempActStep.addStep(1,FALSE);
	END_IF
819:
	IF gICP.HePumValve.Get_Done_Ret() THEN
		tempActStep.addStep(1,FALSE);
	END_IF
820:
	IF gICP.ElectrodeCyl.Get_Done_Ret() THEN
		tempActStep.addStep(20,FALSE);
	ELSE
		IF gICP.ElectrodeCyl.Act_Retract() THEN
			tempActStep.addStep(10,FALSE);
		END_IF
	END_IF
830:
	IF gICP.ElectrodeCyl.Get_Done_Ret() THEN
		tempActStep.addStep(10,FALSE);
	END_IF
840:
	IF gICP.LiftPinCyl.Get_Done_Ret() THEN
		tempActStep.addStep(20,FALSE);
	ELSE
		IF gICP.LiftPinCyl.Act_Retract() THEN
			tempActStep.addStep(10,FALSE);
		END_IF
	END_IF
850:
	IF gICP.LiftPinCyl.Get_Done_Ret() THEN
		tempActStep.addStep(10,FALSE);
	END_IF
860:
	tempActStep.toStep(1000,FALSE);
1000:
	tempActStep.toDoneStep();

60000://Done
	tempActStep.setDoneFlag();
	tempActStep.toZeroStep();
	gWaferMemoryState:=2;
	ups_CX51X0.Act_Wrtie();
	gRunningLog.append('Etching POU Run:----Finish----');
	gRFComControl:=FALSE;
65000://Error
	tempActStep.setErrDoneFlag();
	tempActStep.toZeroStep();
	gRFComControl:=FALSE;
END_CASE
END_METHOD

END_PROGRAM

// ---- POUs/MachinePOU/SemiAutomatic/S_CO_ControlRF.TcPOU
PROGRAM S_CO_ControlRF
VAR_INPUT
	bInit				:BOOL:=FALSE;// 初始化状态 busy/done/errDone
	bTrig				:BOOL:=FALSE;// 执行触发 信号
	bReset				:BOOL:=FALSE;// 报错 复位
	bPause				:BOOL:=FALSE;// 暂停 运行
	bStop				:BOOL:=FALSE;// 停止 运行
	bAbort				:BOOL:=FALSE;// 中止 运行
	
END_VAR
VAR_OUTPUT
	busy				:BOOL;
	done				:BOOL;
	errDone				:BOOL;
	stopDone			:BOOL;
END_VAR
VAR
	actStep				:ActStepBase;
END_VAR
VAR
	i: INT;
	t1:ton;
	t2:ton;
	t3:ton;
	openErrorDelayTon:TON;
	notchoose:BOOL;
	timeOutTime:TIME:= T#60S;
	ventTime:TIME:=T#15S;
END_VAR

busy:=actStep.isBusy();
done:=actStep.isDone();
errDone:=actStep.isError();
actStep.Act_Pause(pause:=bPause);

IF bTrig THEN
	bTrig:=FALSE;
	IF NOT busy THEN
		actStep.Act_ex();
	END_IF
END_IF

//状态复位
IF bInit THEN
	bInit:=FALSE;
	Act_init_status();
END_IF

IF bAbort OR bStop THEN
	bAbort:=FALSE;
	bStop:=FALSE;
	Act_init_status();
	actStep.toZeroStep();
	gShowLogTextTitle:='NON';
	IF gICP.PowerRF.closeCondition AND gICP.SourceRF.closeCondition THEN
		gICP.PowerRF.Act_Close();
		gICP.SourceRF.Act_Close();
		IF gICP.HeINExtRelay THEN
			gICP.HeINValve.Act_Retract();
		END_IF
		gOperatorLog.append('RF_CO_Control CLOSE');
		gICP.PowerRF.co_control:=FALSE;
		gICP.SourceRF.co_control:=FALSE;
	ELSE
		error_Trigger(102);
	END_IF
END_IF
ActionRun(tempActStep:=actStep);
IF NOT gICP.PowerRFOpenRelay AND NOT gICP.SourceRFOpenRelay AND 
	gICP.PowerRF.reflectedpower<1 AND gICP.PowerRF.forwardpower<1 AND
    gICP.SourceRF.reflectedpower<1 AND gICP.SourceRF.forwardpower<1 THEN
	stopDone:=TRUE;
ELSE
	stopDone:=FALSE;
END_IF

(*
---Trigger action
*)
METHOD Act_Ex : BOOL
VAR_INPUT
END_VAR
IF NOT busy THEN
	actStep.Act_ex();
	Act_Ex:=TRUE;
ELSE
	Act_Ex:=FALSE;
END_IF
END_METHOD

(*
---功能: 状态复位 busy/done/errDone;
*)
METHOD Act_Init_Status
VAR_INPUT
END_VAR
actStep.Act_Init();
END_METHOD

METHOD PRIVATE ActionRun
VAR_INPUT
	tempActStep:ITFActStep;
END_VAR
VAR_STAT//此处定义静态变量, 保证每次进入该函数时能够在线监控当前值
	tempStep:DINT;
END_VAR
tempStep:=tempActStep.getStep();
CASE tempStep OF
0:
	IF tempActStep.isEx() THEN
		tempActStep.setBusyFlag();
		tempActStep.toBeginStep();
	END_IF
	t1(IN:= FALSE );
	t2(IN:= FALSE );
	t3(IN:= FALSE );
10:
	IF NOT S_Etching.busy THEN
		gShowLogTextTitle:='CO_Control RF';
	END_IF
	IF gICP.PowerRF.openCondition AND gICP.SourceRF.openCondition THEN
		tempActStep.addStep(10,FALSE);
		gICP.PowerRF.co_control:=TRUE;
		gICP.SourceRF.co_control:=TRUE;
		gRunningLog.append(CONCAT('RF_CO_Control POU Run:',DINT_TO_STRING(tempStep)));
		gRunningLog.append(CONCAT('RF_CO_Control Open,PowerRF POWER:',UDINT_TO_STRING(gICP.PowerRF.setpower)));
		gRunningLog.append(CONCAT('RF_CO_Control Open,SourceRF POWER:',UDINT_TO_STRING(gICP.SourceRF.setpower)));
		IF gCO_ControlRFTimeRemain<>gRFSetTime OR  gCO_ControlRFTimeRemain=0 THEN //  gCO_ControlRFTimeRemain=0代表初次设定
			gRFSetTime:=gRFSetTime;
		ELSE
			gRFSetTime:=gCO_ControlRFTimeRemain;
		END_IF
		gRunningLog.append(CONCAT('RF_CO_Control Open,SET TIME:',UDINT_TO_STRING(gRFSetTime)));
	ELSE
		error_Trigger(100);
	END_IF
20:
	IF gICP.PowerRF.setpower>0 THEN
		IF gICP.PowerRF.Act_Open() THEN
			gRunningLog.append(CONCAT('RF_CO_Control POU Run:',DINT_TO_STRING(tempStep)));
			gRunningLog.append(' PowerRF Open');
			tempActStep.addStep(10,FALSE);
		END_IF
	ELSE
		tempActStep.addStep(20,FALSE);
	END_IF
30:
	IF gICP.PowerRF.Get_Done_Open() THEN
		gRunningLog.append(CONCAT('RF_CO_Control POU Run:',DINT_TO_STRING(tempStep)));
		gRunningLog.append('RF_CO_Control POU Run: PowerRF Open Done');
		tempActStep.addStep(10,FALSE);
	END_IF
	IF gICP.PowerRF.error THEN
		error_Trigger(101);
		tempActStep.toErrDoneStep();
	END_IF
40:
	IF gICP.PowerRF.setpower>0 THEN
		IF gICP.SourceRF.Act_Open() THEN
			gRunningLog.append(CONCAT('RF_CO_Control POU Run:',DINT_TO_STRING(tempStep)));
			gRunningLog.append('RF_CO_Control POU Run: SourceRF Open');
			tempActStep.addStep(10,FALSE);
		END_IF
	ELSE
		tempActStep.addStep(30,FALSE);
	END_IF
50:
	IF gICP.SourceRF.Get_Done_Open() THEN
		gRunningLog.append(CONCAT('RF_CO_Control POU Run:',DINT_TO_STRING(tempStep)));
		gRunningLog.append('RF_CO_Control POU Run: SourceRF Open Done');
		tempActStep.addStep(10,FALSE);
	END_IF
	IF gICP.SourceRF.error THEN
		error_Trigger(101);
		tempActStep.toErrDoneStep();
	END_IF
60:
	openErrorDelayTon(IN:=TRUE,PT:=UDINT_TO_TIME(gCO_ControlRFTime*1000));// 反射调整超时时间
	gCO_ControlRFRMTime:=TIME_TO_UDINT(openErrorDelayTon.ET/1000);
	gCO_ControlRFRMTime:=gCO_ControlRFTime-gCO_ControlRFRMTime;
	IF openErrorDelayTon.Q THEN
		tempActStep.addStep(10,FALSE);
		gCO_ControlRFRMTime:=0;
		openErrorDelayTon(IN:=FALSE);
		RETURN;
	END_IF
	IF gICP.S_MFCMonitFlowNotZero THEN
		error_Trigger(120);
		tempActStep.toErrDoneStep();
		RETURN;
	END_IF
	IF bPause THEN
		gICP.PowerRF.Act_Close();
		gICP.SourceRF.Act_Close();
		gRunningLog.append(CONCAT('RF_CO_Control POU Run:',DINT_TO_STRING(tempStep)));
		gRunningLog.append('RF_CO_Control POU Run: PC Click The Pause Function');
		tempActStep.toErrDoneStep();
	END_IF
70:
	gRunningLog.append(CONCAT('RF_CO_Control POU Run:',DINT_TO_STRING(tempStep)));
	gRunningLog.append('RF_CO_Control POU Run: RF Close');
	gICP.PowerRF.Act_Close();
	gICP.SourceRF.Act_Close();
	tempActStep.addStep(10,FALSE);
80:
	IF gICP.PowerRF.Get_Done_Close() AND gICP.PowerRF.Get_Done_Close()  THEN
		gRunningLog.append(CONCAT('RF_CO_Control POU Run:',DINT_TO_STRING(tempStep)));
		gRunningLog.append('RF_CO_Control POU Run: RF Close Done');
		tempActStep.addStep(10,FALSE);
	END_IF
90:
	tempActStep.toDoneStep();
1000:
	tempActStep.toDoneStep();

60000://Done
	tempActStep.setDoneFlag();
	tempActStep.toZeroStep();
	gICP.PowerRF.co_control:=FALSE;
	gICP.SourceRF.co_control:=FALSE;
	
65000://Error
	tempActStep.setErrDoneFlag();
	tempActStep.toZeroStep();
	gICP.PowerRF.Act_Close();
	gICP.SourceRF.Act_Close();
	gICP.PowerRF.co_control:=FALSE;
	gICP.SourceRF.co_control:=FALSE;
END_CASE
END_METHOD

END_PROGRAM

// ---- POUs/MachinePOU/SemiAutomatic/S_UnLoadWafer.TcPOU
PROGRAM S_UnLoadWafer
VAR_INPUT
	bInit				:BOOL:=FALSE;// 初始化状态 busy/done/errDone
	bTrig				:BOOL:=FALSE;// 执行触发 信号
	bReset				:BOOL:=FALSE;// 报错 复位
	bPause				:BOOL:=FALSE;// 暂停 运行
	bStop				:BOOL:=FALSE;// 停止 运行
	bAbort				:BOOL:=FALSE;// 中止 运行
	
END_VAR
VAR_OUTPUT
	busy				:BOOL;
	done				:BOOL;
	errDone				:BOOL;
END_VAR
VAR
	actStep				:ActStepBase;
END_VAR
VAR
	i: INT;
	t1:ton;
	t2:ton;
	t3:ton;
	notchoose:BOOL;
	timeOutTime:TIME:= T#120S;
	ventTime:TIME:=T#25S;
	ventTimes:INT;
END_VAR

busy:=actStep.isBusy();
done:=actStep.isDone();
errDone:=actStep.isError();
actStep.Act_Pause(pause:=bPause);

IF bTrig THEN
	bTrig:=FALSE;
	IF NOT busy THEN
		actStep.Act_ex();
	END_IF
END_IF

//状态复位
IF bInit THEN
	bInit:=FALSE;
	Act_init_status();
END_IF

IF bAbort OR bStop THEN
	bAbort:=FALSE;
	bStop:=FALSE;
	Act_init_status();
	actStep.toZeroStep();
	gShowLogTextTitle:='NON';
END_IF
ActionRun(tempActStep:=actStep);

(*
---Trigger action
*)
METHOD Act_Ex : BOOL
VAR_INPUT
END_VAR
IF NOT busy THEN
	actStep.Act_ex();
	Act_Ex:=TRUE;
ELSE
	Act_Ex:=FALSE;
END_IF
END_METHOD

(*
---功能: 状态复位 busy/done/errDone;
*)
METHOD Act_Init_Status
VAR_INPUT
END_VAR
actStep.Act_Init();
END_METHOD

METHOD PRIVATE ActionRun
VAR_INPUT
	tempActStep:ITFActStep;
END_VAR
VAR_STAT//此处定义静态变量, 保证每次进入该函数时能够在线监控当前值
	tempStep:DINT;
END_VAR
tempStep:=tempActStep.getStep();
CASE tempStep OF
0:
	IF tempActStep.isEx() THEN
		tempActStep.setBusyFlag();
		tempActStep.toBeginStep();
	END_IF
	t1(IN:= FALSE );
	t2(IN:= FALSE );
	t3(IN:= FALSE );
10:
	gShowLogTextTitle:='UnLoad Wafer';
	IF gRunningState<>RunningStatus.eErrorState THEN
		tempActStep.addStep(10,FALSE);
	ELSE
		error_Trigger(105);
		IF gCtrlMode=ControlMode.eManualCtrMode THEN
			tempActStep.toErrDoneStep();
		END_IF
	END_IF
20:
	IF ControlMode.eManualCtrMode=gCtrlMode THEN
		tempActStep.addStep(40,FALSE);
	ELSIF( ControlMode.eAutoCtrMode=gCtrlMode) THEN
		tempActStep.addStep(40,FALSE);
	ELSE
		tempActStep.toErrDoneStep();
	END_IF
30:
	tempActStep.addStep(10,FALSE);
40:
	tempActStep.addStep(10,TRUE);
50:
	tempActStep.addStep(10,FALSE);
60:
	S_RoughPumping.Act_Init_Status();
	S_RoughPumping.Act_Ex();
	tempActStep.addStep(10,FALSE);
70:
	IF S_RoughPumping.done THEN
		gShowLogTextTitle:='UnLoad Wafer';
		tempActStep.addStep(10,FALSE);
	END_IF
	IF S_RoughPumping.errDone THEN
		tempActStep.toErrDoneStep();
	END_IF
80:
	tempActStep.addStep(20,TRUE);
100:
	IF gWaferMemoryState=1 OR gWaferMemoryState=2 THEN// 腔体有晶圆
		IF NOT gICP.I_WaferCheck THEN
			tempActStep.addStep(10,FALSE);
		ELSE
			error_Trigger(115);
			tempActStep.toErrDoneStep();
		END_IF
	ELSE
		gRunningLog.append(CONCAT('UnLoad Wafer POU Step:',DINT_TO_STRING(tempStep)));
		gRunningLog.append('UnLoad Wafer POU Run:Wafer In Chamber To Vent LoadLock');
		tempActStep.toStep(500,FALSE);// LoadLock有料，则直接判断UnLoad完成（或者衔接无料Vent的过程）
	END_IF
110:
	tempActStep.addStep(5,TRUE);
115:
	IF gICP.GateDoorValve.Act_Retract() AND gICP.VentValve.Act_Retract() THEN
		gRunningLog.append(CONCAT('UnLoad Wafer POU Step:',DINT_TO_STRING(tempStep)));
		gRunningLog.append('UnLoad Wafer POU Run:Gate Door Close And Vent Close');
		tempActStep.addStep(5,FALSE);
	END_IF
120:
	IF gICP.GateDoorValve.Get_Done_Ret() AND gICP.GateDoorRetSensor AND
       gICP.VentValve.Get_Done_Ret() AND NOT gICP.VentExtRelay THEN
	   gRunningLog.append(CONCAT('UnLoad Wafer POU Step:',DINT_TO_STRING(tempStep)));
	   gRunningLog.append('UnLoad Wafer POU Run:Gate Door Close Done And Vent Valve Close Done');
		tempActStep.addStep(10,FALSE);
	END_IF
130:
	IF gICP.ElectrodeCyl.Act_Retract() THEN
		gRunningLog.append(CONCAT('UnLoad Wafer POU Step:',DINT_TO_STRING(tempStep)));
		gRunningLog.append('UnLoad Wafer POU Run:ElectrodeCyl Dowm');
		tempActStep.addStep(10,FALSE);
	END_IF
140:
	IF gICP.ElectrodeCyl.Get_Done_Ret() AND gICP.ElectrodeCylRetSensor THEN
		gRunningLog.append(CONCAT('UnLoad Wafer POU Step:',DINT_TO_STRING(tempStep)));
		gRunningLog.append('UnLoad Wafer POU Run:ElectrodeCyl Dowm Done');
		tempActStep.addStep(10,FALSE);
	END_IF
150:
	tempActStep.addStep(10,FALSE);
160:
	tempActStep.addStep(10,TRUE);
170:
	IF gICP.LiftPinCyl.Act_Extend() THEN
		gRunningLog.append(CONCAT('UnLoad Wafer POU Step:',DINT_TO_STRING(tempStep)));
		gRunningLog.append('UnLoad Wafer POU Run:LiftPinCyl UP');
		tempActStep.addStep(10,FALSE);
	END_IF
180:
	IF gICP.LiftPinCyl.Get_Done_Ext() AND gICP.LiftPinExtSensor THEN
		gRunningLog.append(CONCAT('UnLoad Wafer POU Step:',DINT_TO_STRING(tempStep)));
		gRunningLog.append('UnLoad Wafer POU Run:LiftPinCyl UP Down');
		tempActStep.addStep(10,FALSE);
	END_IF
190:
	t1(IN:=TRUE,PT:=T#1S);
	IF t1.Q THEN
		t1(IN:= FALSE );
		t2(IN:= FALSE );
		t3(IN:= FALSE );
		tempActStep.addStep(10,FALSE);
	END_IF
200:
	tempActStep.addStep(10,FALSE);
210:
	tempActStep.addStep(10,TRUE);
220:
	IF NOT gICP.VentExtRelay AND gICP.ForlinLineValveExtRelay AND NOT gICP.RoughValveExtRelay THEN
		tempActStep.addStep(10,FALSE);
	ELSE
		error_Trigger(105);
		tempActStep.toStep(210,FALSE);
	END_IF
230://////////////准备破LoadLock
	IF gICP.LoadLockGauge.outputValue<gRoughtPumVaccum THEN // LL 真空满足
		IF NOT gICP.LoadLockGauge.error AND gICP.PDV.Act_Retract()  THEN
			tempActStep.toStep(340,FALSE);
			gRunningLog.append(CONCAT('UnLoad Wafer POU Step:',DINT_TO_STRING(tempStep)));
			gRunningLog.append(CONCAT('UnLoad Wafer POU Run:LL Pressure Arrive ',REAL_TO_STRING(gICP.LoadLockGauge.outputValue)));
		ELSE
			error_Trigger(105);
			tempActStep.toStep(210,FALSE);
		END_IF
	ELSE
		tempActStep.addStep(10,FALSE);
	END_IF
240:
	tempActStep.addStep(2,TRUE);
242:
	IF gICP.ForlinLineValve.Act_Retract() AND gICP.PDV.Act_Retract() THEN
		tempActStep.addStep(2,FALSE);
	END_IF
244:
	IF gICP.ForlinLineValve.Get_Done_Ret() AND (gICP.PDVCloseSensor OR gICP.PDV.Get_Done_Ret()) THEN
		tempActStep.addStep(2,FALSE);
	END_IF
246:
	tempActStep.addStep(4,TRUE);
250:
	IF gICP.SlowPummingValve.Act_Extend() AND gICP.FastPummingValve.Act_Retract() THEN
		gRunningLog.append(CONCAT('UnLoad Wafer POU Step:',DINT_TO_STRING(tempStep)));
		gRunningLog.append('UnLoad Wafer POU Run:SlowPummingValve Open and FastPummingValve Close');
		tempActStep.addStep(10,FALSE);
	END_IF
260:
	IF gICP.SlowPummingValve.Get_Done_Ext() AND gICP.FastPummingValve.Get_Done_Ret() THEN
		gRunningLog.append(CONCAT('UnLoad Wafer POU Step:',DINT_TO_STRING(tempStep)));
		gRunningLog.append('UnLoad Wafer POU Run:SlowPummingValve Open Done and FastPummingValve Close Done');
		tempActStep.addStep(10,FALSE);
	END_IF
270:
	t2(IN:=gICP.LoadLockGauge.outputValue<gLoadLockPumSVaccum,PT:=T#2S);
	IF t2.Q THEN
		t1(IN:= FALSE );
		t2(IN:= FALSE );
		t3(IN:= FALSE );
		gRunningLog.append(CONCAT('UnLoad Wafer POU Step:',DINT_TO_STRING(tempStep)));
		gRunningLog.append(CONCAT('UnLoad Wafer POU Run:LL Pressure Arrive ',REAL_TO_STRING(gICP.LoadLockGauge.outputValue)));
		tempActStep.addStep(10,FALSE);
	END_IF
280:
	IF gICP.SlowPummingValve.Act_Retract() AND gICP.FastPummingValve.Act_Extend() THEN
		gRunningLog.append(CONCAT('UnLoad Wafer POU Step:',DINT_TO_STRING(tempStep)));
		gRunningLog.append('UnLoad Wafer POU Run:SlowPummingValve Close and FastPummingValve Open');
		tempActStep.addStep(10,FALSE);
	END_IF
290:
	IF gICP.SlowPummingValve.Get_Done_Ret() AND gICP.FastPummingValve.Get_Done_Ext() THEN
		gRunningLog.append(CONCAT('UnLoad Wafer POU Step:',DINT_TO_STRING(tempStep)));
		gRunningLog.append('UnLoad Wafer POU Run:SlowPummingValve Close Done and FastPummingValve Open Done');
		tempActStep.addStep(10,FALSE);
	END_IF
300:
	t2(IN:=gICP.LoadLockGauge.outputValue<gRoughtPumVaccum,PT:=T#2S);
	IF t2.Q THEN
		t1(IN:= FALSE );
		t2(IN:= FALSE );
		t3(IN:= FALSE );
		gRunningLog.append(CONCAT('UnLoad Wafer POU Step:',DINT_TO_STRING(tempStep)));
		gRunningLog.append(CONCAT('UnLoad Wafer POU Run:LL Pressure Arrive ',REAL_TO_STRING(gICP.LoadLockGauge.outputValue)));
		tempActStep.addStep(10,FALSE);
	END_IF
310:
	tempActStep.addStep(10,TRUE);
320:
	IF gICP.SlowPummingValve.Act_Retract() AND gICP.FastPummingValve.Act_Retract() AND gICP.PDV.Act_Retract() THEN
		gRunningLog.append(CONCAT('UnLoad Wafer POU Step:',DINT_TO_STRING(tempStep)));
		gRunningLog.append('UnLoad Wafer POU Run:SlowPummingValve Close | FastPummingValve Close | PDV Open');
		tempActStep.addStep(10,FALSE);
	END_IF
330:
	IF gICP.SlowPummingValve.Get_Done_Ret() AND gICP.FastPummingValve.Get_Done_Ret() AND (gICP.PDV.Get_Done_Ret() OR gICP.PDVCloseSensor) THEN
		gRunningLog.append(CONCAT('UnLoad Wafer POU Step:',DINT_TO_STRING(tempStep)));
		gRunningLog.append('UnLoad Wafer POU Run:SlowPummingValve Close Done | FastPummingValve Close Done | PDV Open Done');
		tempActStep.addStep(10,FALSE);
	END_IF
340:
	IF (gICP.PDV.Get_Done_Ret() OR gICP.PDVCloseSensor) THEN
		tempActStep.addStep(10,TRUE);
	END_IF
350:
	IF gICP.GateDoorValve.Act_Extend() THEN
		gRunningLog.append(CONCAT('UnLoad Wafer POU Step:',DINT_TO_STRING(tempStep)));
		gRunningLog.append('UnLoad Wafer POU Run:Gate Door Open');
		tempActStep.addStep(5,FALSE);
	END_IF
355:
	IF gICP.GateDoorValve.Get_Done_Ext() AND gICP.GateDoorExtSensor THEN
		gRunningLog.append(CONCAT('UnLoad Wafer POU Step:',DINT_TO_STRING(tempStep)));
		gRunningLog.append('UnLoad Wafer POU Run:Gate Door Open Done');
		tempActStep.addStep(5,FALSE);
	END_IF
360:
	IF gICP.HeMFC_ActFlow<1 AND gICP.HeCheckGaugeReal<1 AND NOT gICP.HeINExtRelay AND NOT gICP.HePumExtRelay THEN
		tempActStep.addStep(1,FALSE);
	ELSE
		tempActStep.addStep(10,FALSE);
	END_IF
361:
	tempActStep.addStep(1,TRUE);
362:
	IF gICP.HeINValve.Act_Retract() THEN
		tempActStep.addStep(1,FALSE);
	END_IF
363:
	IF gICP.HeINValve.Get_Done_Ret() THEN
		tempActStep.addStep(1,FALSE);
	END_IF
364:
	tempActStep.addStep(1,TRUE);
365:
	IF gICP.HePumValve.Act_Extend() THEN
		tempActStep.addStep(1,FALSE);
	END_IF
366:
	IF gICP.HePumValve.Get_Done_Ext() THEN
		tempActStep.addStep(1,FALSE);
	END_IF
367:
	t2(IN:=TRUE ,PT:=T#2S);
	IF t2.Q THEN
		t1(IN:= FALSE );
		t2(IN:= FALSE );
		t3(IN:= FALSE );
		tempActStep.addStep(1,FALSE);
	END_IF
368:
	t1(IN:=gICP.HeMFC_ActFlow<1 AND gICP.HeCheckGaugeReal<1 ,PT:=T#2S);
	IF t1.Q THEN
		t1(IN:= FALSE );
		t2(IN:= FALSE );
		t3(IN:= FALSE );
		gICP.HePumValve.Act_Retract();
		tempActStep.addStep(2,FALSE);
	END_IF
370:
	IF gICP.ElectrodeCyl.Act_Retract() AND gICP.HePumValve.Get_Done_Ret() THEN
		gRunningLog.append(CONCAT('UnLoad Wafer POU Step:',DINT_TO_STRING(tempStep)));
		gRunningLog.append('UnLoad Wafer POU Run:ElectrodeCyl Down');
		tempActStep.addStep(2,FALSE);
	END_IF
372:
	IF gICP.ElectrodeCyl.Get_Done_Ret() THEN
		gRunningLog.append(CONCAT('UnLoad Wafer POU Step:',DINT_TO_STRING(tempStep)));
		gRunningLog.append('UnLoad Wafer POU Run:ElectrodeCyl Down Done');
		tempActStep.addStep(2,FALSE);
	END_IF
374:
	tempActStep.addStep(2,TRUE);
376:
	IF gICP.LiftPinCyl.Act_Extend() THEN
		gRunningLog.append(CONCAT('UnLoad Wafer POU Step:',DINT_TO_STRING(tempStep)));
		gRunningLog.append('UnLoad Wafer POU Run:LiftPinCyl UP');
		tempActStep.addStep(2,FALSE);
	END_IF
378:
	IF gICP.LiftPinCyl.Get_Done_Ext() THEN
		gRunningLog.append(CONCAT('UnLoad Wafer POU Step:',DINT_TO_STRING(tempStep)));
		gRunningLog.append('UnLoad Wafer POU Run:LiftPinCyl UP Done');
		tempActStep.addStep(1,FALSE);
	END_IF
379:
	tempActStep.addStep(1,TRUE);
380:
	tempActStep.addStep(20,FALSE);
400:
	IF gICP.ARM.Act_IN_Auto() THEN
		gRunningLog.append(CONCAT('UnLoad Wafer POU Step:',DINT_TO_STRING(tempStep)));
		gRunningLog.append('UnLoad Wafer POU Run:ARM IN');
		tempActStep.addStep(10,FALSE);
	END_IF
410:
	IF NOT gICP.I_ARMHome THEN// 手臂当前不应该在原点位置
		tempActStep.addStep(10,FALSE);
	END_IF
420:
	t1(IN:=gICP.ARM.Get_Done_IN() AND NOT gICP.ARM.busy AND ABS(gICP.ARM.actpos-gARMPosition)<=1 ,PT:=T#2S);
	IF t1.Q THEN
		t1(IN:= FALSE );
		t2(IN:= FALSE );
		t3(IN:= FALSE );
		gRunningLog.append(CONCAT('UnLoad Wafer POU Step:',DINT_TO_STRING(tempStep)));
		gRunningLog.append('UnLoad Wafer POU Run:ARM IN Done');
		tempActStep.addStep(10,FALSE);
		RETURN;
	END_IF
	t2(IN:=TRUE,PT:=T#20S);
	IF t2.Q THEN
		t1(IN:= FALSE );
		t2(IN:= FALSE );
		t3(IN:= FALSE );
		error_Trigger(114);
		tempActStep.toStep(379,FALSE);
		RETURN;
	END_IF
430:
	tempActStep.addStep(10,TRUE);
440:
	IF gICP.LiftPinCyl.Act_Retract() THEN
		gRunningLog.append(CONCAT('UnLoad Wafer POU Step:',DINT_TO_STRING(tempStep)));
		gRunningLog.append('UnLoad Wafer POU Run:LiftPinCyl Down');
		tempActStep.addStep(10,FALSE);
	END_IF
450:
	IF gICP.LiftPinCyl.Get_Done_Ret() AND gICP.LiftPinRetSensor THEN
		gRunningLog.append(CONCAT('UnLoad Wafer POU Step:',DINT_TO_STRING(tempStep)));
		gRunningLog.append('UnLoad Wafer POU Run:LiftPinCyl Down Done');
		// 记忆状态更新
		gWaferMemoryState:=0;
		ups_CX51X0.Act_Wrtie();
		tempActStep.addStep(10,FALSE);
	END_IF
460:
	tempActStep.addStep(10,TRUE);
470:
	IF gICP.ARM.Act_HOME_Auto() THEN
		gRunningLog.append(CONCAT('UnLoad Wafer POU Step:',DINT_TO_STRING(tempStep)));
		gRunningLog.append('UnLoad Wafer POU Run:ARM Home');
		tempActStep.addStep(10,FALSE);
	END_IF
480:
	IF gICP.ARM.Get_Done_HOME() AND gICP.I_ARMHome AND ABS(gICP.ARM.actpos-0)<=1 AND NOT gICP.ARM.busy THEN// 手臂当前不应该在原点位置
		gRunningLog.append(CONCAT('UnLoad Wafer POU Step:',DINT_TO_STRING(tempStep)));
		gRunningLog.append('UnLoad Wafer POU Run:ARM Home Done');
		tempActStep.addStep(10,FALSE);
	END_IF
490:
	t2(IN:=TRUE,PT:=T#2S);
	IF t2.Q THEN
		t1(IN:= FALSE );
		t2(IN:= FALSE );
		t3(IN:= FALSE );
		tempActStep.addStep(10,FALSE);
		RETURN;
	END_IF
500:
	ventTimes:=1;
	tempActStep.addStep(10,TRUE);
510:
	IF gICP.GateDoorValve.Act_Retract() THEN
		gRunningLog.append(CONCAT('UnLoad Wafer POU Step:',DINT_TO_STRING(tempStep)));
		gRunningLog.append('UnLoad Wafer POU Run:GateDoorValve Close');
		tempActStep.addStep(10,FALSE);
	END_IF
520:
	IF gICP.GateDoorValve.Get_Done_Ret() AND gICP.GateDoorRetSensor THEN
		gRunningLog.append(CONCAT('UnLoad Wafer POU Step:',DINT_TO_STRING(tempStep)));
		gRunningLog.append('UnLoad Wafer POU Run:GateDoorValve Close Done');
		tempActStep.addStep(10,FALSE);
	END_IF
530:
	tempActStep.addStep(10,TRUE);
540:
	IF  gICP.GateDoorValve.Act_Retract() AND 
	    gICP.SlowPummingValve.Act_Retract() AND 
	    gICP.FastPummingValve.Act_Retract() THEN
		tempActStep.addStep(10,FALSE);
	END_IF
550:
	IF gICP.GateDoorValve.Get_Done_Ret() AND gICP.GateDoorRetSensor AND
	   gICP.SlowPummingValve.Get_Done_Ret() AND NOT gICP.SlowPummingExtRelay AND
	   gICP.FastPummingValve.Get_Done_Ret() AND NOT gICP.FastPummingExtRelay THEN
		tempActStep.addStep(10,FALSE);
	END_IF
560:
	IF gICP.VentValve.Act_Extend() THEN
		gRunningLog.append(CONCAT('UnLoad Wafer POU Step:',DINT_TO_STRING(tempStep)));
		gRunningLog.append('UnLoad Wafer POU Run:VentValve Open');
		tempActStep.addStep(10,FALSE);
	END_IF
570:
	IF gICP.VentValve.Get_Done_Ext() THEN
		gRunningLog.append(CONCAT('UnLoad Wafer POU Step:',DINT_TO_STRING(tempStep)));
		gRunningLog.append('UnLoad Wafer POU Run:VentValve Open Done');
		tempActStep.addStep(10,FALSE);
	END_IF
580:
	t2(IN:=gICP.LoadLockGauge.outputValue>gATMPressure,PT:=ventTime/ventTimes);
	IF t2.Q OR NOT gICP.I_LLSwitch THEN
		t1(IN:= FALSE );
		t2(IN:= FALSE );
		t3(IN:= FALSE );
		gRunningLog.append(CONCAT('UnLoad Wafer POU Step:',DINT_TO_STRING(tempStep)));
		gRunningLog.append(CONCAT('UnLoad Wafer POU Run:LL Pressure Arrive ',REAL_TO_STRING(gICP.LoadLockGauge.outputValue)));
		tempActStep.addStep(10,FALSE);
	END_IF
590:
	tempActStep.addStep(10,TRUE);
600:
	IF gICP.VentValve.Act_Retract() THEN
		gRunningLog.append(CONCAT('UnLoad Wafer POU Step:',DINT_TO_STRING(tempStep)));
		gRunningLog.append('UnLoad Wafer POU Run:VentValve Close');
		tempActStep.addStep(10,FALSE);
	END_IF
610:
	IF gICP.VentValve.Get_Done_Ret() THEN
		gRunningLog.append(CONCAT('UnLoad Wafer POU Step:',DINT_TO_STRING(tempStep)));
		gRunningLog.append('UnLoad Wafer POU Run:VentValve Close Done');
		tempActStep.addStep(10,FALSE);
	END_IF
620:
	t1(IN:=TRUE,PT:=T#1S);
	IF t1.Q THEN
		t1(IN:= FALSE );
		t2(IN:= FALSE );
		t3(IN:= FALSE );
		gRunningLog.append('UnLoad Wafer POU Run:Wait for the wafer to be removed');
		tempActStep.addStep(10,FALSE);
	END_IF
630:
	t2(IN:=NOT gICP.I_WaferCheck AND gICP.I_LLSwitch,PT:=T#1S);// 拿走晶圆，且关上盖子
	IF t2.Q THEN
		t1(IN:= FALSE );
		t2(IN:= FALSE );
		t3(IN:= FALSE );
		gRunningLog.append(CONCAT('UnLoad Wafer POU Step:',DINT_TO_STRING(tempStep)));
		gRunningLog.append('UnLoad Wafer POU Run:Wafer tack out and close LL');
		tempActStep.addStep(10,FALSE);
		RETURN;
	END_IF
	t3(IN:=TRUE,PT:=timeOutTime);
	IF t3.Q THEN
		error_Trigger(114);
		ventTimes:=3;
		tempActStep.toStep(530,FALSE);
	END_IF
640:
	IF gICP.ForlinLineValve.Act_Extend() THEN
		gRunningLog.append(CONCAT('UnLoad Wafer POU Step:',DINT_TO_STRING(tempStep)));
		gRunningLog.append('UnLoad Wafer POU Run:ForLineValve Open');
		tempActStep.addStep(10,FALSE);
	END_IF
650:
	IF gICP.ForlinLineValve.Get_Done_Ext() THEN
		gRunningLog.append(CONCAT('UnLoad Wafer POU Step:',DINT_TO_STRING(tempStep)));
		gRunningLog.append('UnLoad Wafer POU Run:ForLineValve Open Done');
		tempActStep.addStep(10,FALSE);
	END_IF
660:
	tempActStep.addStep(10,TRUE);
670:
	IF gICP.PDV.Act_Open() THEN
		gRunningLog.append(CONCAT('UnLoad Wafer POU Step:',DINT_TO_STRING(tempStep)));
		gRunningLog.append('UnLoad Wafer POU Run:PDV Open');
		tempActStep.addStep(10,FALSE);
	END_IF
680:
	IF gICP.PDV.Get_Done_Ext() OR gICP.PDVOpenSensor THEN
		gRunningLog.append(CONCAT('UnLoad Wafer POU Step:',DINT_TO_STRING(tempStep)));
		gRunningLog.append('UnLoad Wafer POU Run:PDV Open Done');
		tempActStep.addStep(10,FALSE);
	END_IF
690:
	// 记忆状态更新
	gWaferMemoryState:=0;
	ups_CX51X0.Act_Wrtie();
	gRunningLog.append(CONCAT('UnLoad Wafer POU Step:',DINT_TO_STRING(tempStep)));
	gRunningLog.append('UnLoad Wafer POU Run:----Finish----');
	tempActStep.toDoneStep();
1000:
	tempActStep.toDoneStep();

60000://Done
	tempActStep.setDoneFlag();
	tempActStep.toZeroStep();
	
65000://Error
	tempActStep.setErrDoneFlag();
	tempActStep.toZeroStep();
	IF gICP.VentExtRelay THEN
		gICP.VentValve.Act_Retract();
	END_IF
END_CASE
END_METHOD

END_PROGRAM

// ---- POUs/MachinePOU/SemiAutomatic/S_LoadLockPumping.TcPOU
PROGRAM S_LoadLockPumping
VAR_INPUT
	bInit				:BOOL:=FALSE;// 初始化状态 busy/done/errDone
	bTrig				:BOOL:=FALSE;// 执行触发 信号
	bReset				:BOOL:=FALSE;// 报错 复位
	bPause				:BOOL:=FALSE;// 暂停 运行
	bStop				:BOOL:=FALSE;// 停止 运行
	bAbort				:BOOL:=FALSE;// 中止 运行
	
END_VAR
VAR_OUTPUT
	busy				:BOOL;
	done				:BOOL;
	errDone				:BOOL;
END_VAR
VAR
	actStep				:ActStepBase;
END_VAR
VAR
	i: INT;
	t1:ton;
	t2:ton;
	t3:ton;
	notchoose:BOOL;
	timeOutTime:TIME:=T#120S;
	safecheckTime:TIME:=T#1S;
	pdvOpenflag:BOOL;
	forelineOpenflag:BOOL;
END_VAR

busy:=actStep.isBusy();
done:=actStep.isDone();
errDone:=actStep.isError();
actStep.Act_Pause(pause:=bPause);

IF bTrig THEN
	bTrig:=FALSE;
	IF NOT busy THEN
		actStep.Act_ex();
	END_IF
END_IF

//状态复位
IF bInit THEN
	bInit:=FALSE;
	Act_init_status();
END_IF

IF bAbort OR bStop THEN
	bAbort:=FALSE;
	bStop:=FALSE;
	Act_init_status();
	actStep.toZeroStep();
	gShowLogTextTitle:='NON';
END_IF
ActionRun(tempActStep:=actStep);

(*
---Trigger action
*)
METHOD Act_Ex : BOOL
VAR_INPUT
END_VAR
IF NOT busy THEN
	actStep.Act_ex();
	Act_Ex:=TRUE;
ELSE
	Act_Ex:=FALSE;
END_IF
END_METHOD

(*
---功能: 状态复位 busy/done/errDone;
*)
METHOD Act_Init_Status
VAR_INPUT
END_VAR
actStep.Act_Init();
END_METHOD

METHOD PRIVATE ActionRun
VAR_INPUT
	tempActStep:ITFActStep;
END_VAR
VAR
END_VAR
VAR_STAT//此处定义静态变量, 保证每次进入该函数时能够在线监控当前值
	tempStep:DINT;
END_VAR
tempStep:=tempActStep.getStep();
CASE tempStep OF
0:
	IF tempActStep.isEx() THEN
		tempActStep.setBusyFlag();
		tempActStep.toBeginStep();
	END_IF
	t1(IN:= FALSE );
	t2(IN:= FALSE );
	t3(IN:= FALSE );
10:
	gShowLogTextTitle:='Load Lock Pumping';
	IF gRunningState<>RunningStatus.eErrorState THEN
		tempActStep.addStep(10,FALSE);
	ELSE
		error_Trigger(105);
		IF gCtrlMode=ControlMode.eManualCtrMode THEN
			tempActStep.toErrDoneStep();
		END_IF
	END_IF
20:
	IF NOT gICP.ForeLineGauge.error AND gICP.ForeLineGauge.outputValue<gRoughtPumVaccum*10 THEN
		tempActStep.addStep(10,FALSE);
	ELSE
		error_Trigger(107);
		IF gCtrlMode=ControlMode.eManualCtrMode THEN
			tempActStep.toErrDoneStep();
		END_IF
	END_IF
30:
	IF gICP.ForlinLineValveExtRelay THEN
		forelineOpenflag:=TRUE;
	ELSE
		forelineOpenflag:=FALSE;
	END_IF
	IF gICP.PDVOpenSensor THEN
		pdvOpenflag:=TRUE;
	ELSE
		pdvOpenflag:=FALSE;
	END_IF
	tempActStep.toStep(100,FALSE);
100:
	tempActStep.addStep(10,TRUE);
110:
	IF NOT gRoughRemain THEN
		S_RoughPumping.Act_Init_Status();
		S_RoughPumping.Act_Ex();
		tempActStep.addStep(10,FALSE);
	ELSE
		tempActStep.toStep(160,FALSE);
	END_IF
120:
	IF S_RoughPumping.done THEN
		gShowLogTextTitle:='Load Lock Pumping';
		tempActStep.addStep(10,FALSE);
	END_IF
	IF S_RoughPumping.errDone THEN
		tempActStep.toStep(100,FALSE);
	END_IF
130:
	tempActStep.addStep(10,FALSE);
140:
	IF gICP.ForlinLineValve.Act_Retract() AND gICP.PDV.Act_Retract() THEN
		gRunningLog.append(CONCAT('LLPumping POU Run:',DINT_TO_STRING(tempStep)));
		gRunningLog.append('LLPumping POU Run:ForeLineValve And PDV Close');
		tempActStep.addStep(10,FALSE);
	END_IF
150:
	IF gICP.ForlinLineValve.Get_Done_Ret() AND gICP.PDV.Get_Done_Ret() AND gICP.PDVCloseSensor THEN
		gRunningLog.append(CONCAT('LLPumping POU Run:',DINT_TO_STRING(tempStep)));
		gRunningLog.append('LLPumping POU Run:ForeLineValve And PDV Close Done');
		tempActStep.toStep(200,FALSE);
	END_IF
160:
	S_ActuatorRecoveryPOU.Act_Init_Status();
	S_ActuatorRecoveryPOU.Act_Ex();
	tempActStep.addStep(10,FALSE);
170:
	IF S_ActuatorRecoveryPOU.done THEN
		tempActStep.addStep(10,FALSE);
	END_IF
180:
	tempActStep.addStep(10,FALSE);
190:
	tempActStep.addStep(10,FALSE);
200:
	tempActStep.addStep(10,TRUE);
210:
	IF gICP.GateDoorValve.Get_Done_Ret() AND gICP.GateDoorRetSensor AND
		gICP.VentValve.Get_Done_Ret() AND NOT gICP.VentExtRelay AND
		gICP.SlowPummingValve.Get_Done_Ret() AND NOT gICP.SlowPummingExtRelay AND
		gICP.FastPummingValve.Get_Done_Ret() AND NOT gICP.FastPummingExtRelay AND
		gICP.ForlinLineValve.Get_Done_Ret() AND NOT gICP.ForlinLineValveExtRelay AND
		gICP.RoughValve.Get_Done_Ret() AND NOT gICP.RoughValveExtRelay  THEN
		tempActStep.addStep(10,FALSE);		
	END_IF
220:
	IF gICP.SlowPummingValve.Act_Extend() THEN
		gRunningLog.append(CONCAT('LLPumping POU Run:',DINT_TO_STRING(tempStep)));
		gRunningLog.append('LLPumping POU Run:SlowPummingValve Open');
		tempActStep.addStep(10,FALSE);
	END_IF
230:
	IF gICP.SlowPummingValve.Get_Done_Ext() THEN
		gRunningLog.append(CONCAT('LLPumping POU Run:',DINT_TO_STRING(tempStep)));
		gRunningLog.append('LLPumping POU Run:SlowPummingValve Open Done');
		tempActStep.addStep(10,FALSE);
	END_IF
240:
	t2(IN:= gICP.LoadLockGauge.outputValue<gLoadLockPumSVaccum,PT:=safecheckTime );
	IF t2.Q THEN
		t1(IN:= FALSE );
		t2(IN:= FALSE );
		t3(IN:= FALSE );
		gRunningLog.append(CONCAT('LLPumping POU Run:',DINT_TO_STRING(tempStep)));
		gRunningLog.append(CONCAT('LLPumping POU Run: Slow Pump Pressure Arrive ',REAL_TO_STRING(gICP.LoadLockGauge.outputValue)));
		tempActStep.addStep(10,FALSE);
		RETURN;
	END_IF
	t1(IN:= TRUE,PT:=timeOutTime );
	IF t1.Q THEN
		t1(IN:= FALSE );
		t2(IN:= FALSE );
		t3(IN:= FALSE );
		error_Trigger(122);
		RETURN;
	END_IF
250:
	tempActStep.addStep(10,TRUE);
260:
	IF gICP.SlowPummingValve.Act_Retract() THEN
		gRunningLog.append(CONCAT('LLPumping POU Run:',DINT_TO_STRING(tempStep)));
		gRunningLog.append('LLPumping POU Run:SlowPummingValve Close');
		tempActStep.addStep(10,FALSE);
	END_IF
270:
	IF gICP.SlowPummingValve.Get_Done_Ret() THEN
		gRunningLog.append(CONCAT('LLPumping POU Run:',DINT_TO_STRING(tempStep)));
		gRunningLog.append('LLPumping POU Run:SlowPummingValve Close Done');
		tempActStep.addStep(10,FALSE);
	END_IF
280:
	t3(IN:=TRUE,PT:=T#1S);
	IF t3.Q THEN
		t1(IN:= FALSE );
		t2(IN:= FALSE );
		t3(IN:= FALSE );
		gRunningLog.append(CONCAT('LLPumping POU Run:',DINT_TO_STRING(tempStep)));
		gRunningLog.append(CONCAT('LLPumping POU Run: Fast Pump Pressure Arrive ',REAL_TO_STRING(gICP.LoadLockGauge.outputValue)));
		tempActStep.addStep(10,FALSE);
	END_IF
290:
	tempActStep.addStep(10,TRUE);
300:
	IF gICP.FastPummingValve.Act_Extend() THEN
		gRunningLog.append(CONCAT('LLPumping POU Run:',DINT_TO_STRING(tempStep)));
		gRunningLog.append('LLPumping POU Run:FastPummingValve Open');
		tempActStep.addStep(10,FALSE);
	END_IF
310:
	IF gICP.FastPummingValve.Get_Done_Ext() THEN
		gRunningLog.append(CONCAT('LLPumping POU Run:',DINT_TO_STRING(tempStep)));
		gRunningLog.append('LLPumping POU Run:FastPummingValve Open Done');
		tempActStep.addStep(10,FALSE);
	END_IF
320:
	t2(IN:= gICP.LoadLockGauge.outputValue<gRoughtPumVaccum*10,PT:=safecheckTime );
	IF t2.Q THEN
		t1(IN:= FALSE );
		t2(IN:= FALSE );
		t3(IN:= FALSE );
		gRunningLog.append(CONCAT('LLPumping POU Run:',DINT_TO_STRING(tempStep)));
		gRunningLog.append(CONCAT('LLPumping POU Run: Fast Pump Pressure Arrive ',REAL_TO_STRING(gICP.LoadLockGauge.outputValue)));
		tempActStep.addStep(10,FALSE);
		RETURN;
	END_IF
	t1(IN:= TRUE,PT:=timeOutTime );
	IF t1.Q THEN
		t1(IN:= FALSE );
		t2(IN:= FALSE );
		t3(IN:= FALSE );
		error_Trigger(122);
		RETURN;
	END_IF
330:
	tempActStep.addStep(10,TRUE);
340:
	IF gICP.FastPummingValve.Act_Retract() THEN
		gRunningLog.append(CONCAT('LLPumping POU Run:',DINT_TO_STRING(tempStep)));
		gRunningLog.append('LLPumping POU Run:FastPummingValve Close');
		tempActStep.addStep(10,FALSE);
	END_IF
350:
	IF gICP.FastPummingValve.Get_Done_Ret() THEN
		gRunningLog.append(CONCAT('LLPumping POU Run:',DINT_TO_STRING(tempStep)));
		gRunningLog.append('LLPumping POU Run:FastPummingValve Close Done');
		tempActStep.addStep(10,FALSE);
	END_IF
360:
	t3(IN:=TRUE,PT:=T#2S);
	IF t3.Q THEN
		t1(IN:= FALSE );
		t2(IN:= FALSE );
		t3(IN:= FALSE );
		tempActStep.addStep(10,FALSE);
	END_IF
370:
	tempActStep.addStep(10,TRUE);
380:
	IF forelineOpenflag THEN
		IF gICP.ForlinLineValve.Act_Extend() THEN
			gRunningLog.append(CONCAT('LLPumping POU Run:',DINT_TO_STRING(tempStep)));
			gRunningLog.append('LLPumping POU Run:ForeLineValve Open');
			tempActStep.addStep(10,FALSE);
		END_IF
	ELSE
		tempActStep.toStep(400,FALSE);
	END_IF
	
390:
	IF gICP.ForlinLineValve.Get_Done_Ext() THEN
		gRunningLog.append(CONCAT('LLPumping POU Run:',DINT_TO_STRING(tempStep)));
		gRunningLog.append('LLPumping POU Run:ForeLineValve Open Done');
		tempActStep.addStep(10,FALSE);
	END_IF
400:
	tempActStep.addStep(10,TRUE);
//465:
//	IF gICP.PDV.Act_ChangePos() THEN
//		tempActStep.addStep(2,FALSE);
//	END_IF
//467:
//	IF gICP.PDV.PosMode THEN
//		tempActStep.addStep(3,FALSE);
//	END_IF
410:
	IF pdvOpenflag THEN
		IF gICP.PDV.Act_Open() THEN
			gRunningLog.append(CONCAT('LLPumping POU Run:',DINT_TO_STRING(tempStep)));
			gRunningLog.append('LLPumping POU Run:PDV Open');
			tempActStep.addStep(10,FALSE);
		END_IF
	ELSE
		tempActStep.toStep(1000,FALSE);
	END_IF
	
420:
	IF gICP.PDV.Get_Done_Ext() OR gICP.PDVCloseSensor THEN
		gRunningLog.append(CONCAT('LLPumping POU Run:',DINT_TO_STRING(tempStep)));
		gRunningLog.append('LLPumping POU Run:PDV Open Done');
		tempActStep.addStep(10,FALSE);
	END_IF
430:
	tempActStep.toStep(1000,FALSE);
1000:
	tempActStep.toDoneStep();

60000://Done
	tempActStep.setDoneFlag();
	tempActStep.toZeroStep();
	
65000://Error
	tempActStep.setErrDoneFlag();
	tempActStep.toZeroStep();
END_CASE
END_METHOD

END_PROGRAM

// ---- POUs/MachinePOU/SemiAutomatic/S_LoadLockVent.TcPOU
PROGRAM S_LoadLockVent
VAR_INPUT
	bInit				:BOOL:=FALSE;// 初始化状态 busy/done/errDone
	bTrig				:BOOL:=FALSE;// 执行触发 信号
	bReset				:BOOL:=FALSE;// 报错 复位
	bPause				:BOOL:=FALSE;// 暂停 运行
	bStop				:BOOL:=FALSE;// 停止 运行
	bAbort				:BOOL:=FALSE;// 中止 运行
	
END_VAR
VAR_OUTPUT
	busy				:BOOL;
	done				:BOOL;
	errDone				:BOOL;
END_VAR
VAR
	actStep				:ActStepBase;
END_VAR
VAR
	i: INT;
	t1:ton;
	t2:ton;
	t3:ton;
	notchoose:BOOL;
	timeOutTime:TIME:=T#120S;
	safecheckTime:TIME:=T#1S;
	pdvOpenflag:BOOL;
	forelineOpenflag:BOOL;
END_VAR

busy:=actStep.isBusy();
done:=actStep.isDone();
errDone:=actStep.isError();
actStep.Act_Pause(pause:=bPause);

IF bTrig THEN
	bTrig:=FALSE;
	IF NOT busy THEN
		actStep.Act_ex();
	END_IF
END_IF

//状态复位
IF bInit THEN
	bInit:=FALSE;
	Act_init_status();
END_IF

IF bAbort OR bStop THEN
	bAbort:=FALSE;
	bStop:=FALSE;
	Act_init_status();
	actStep.toZeroStep();
	gShowLogTextTitle:='NON';
END_IF
ActionRun(tempActStep:=actStep);

(*
---Trigger action
*)
METHOD Act_Ex : BOOL
VAR_INPUT
END_VAR
IF NOT busy THEN
	actStep.Act_ex();
	Act_Ex:=TRUE;
ELSE
	Act_Ex:=FALSE;
END_IF
END_METHOD

(*
---功能: 状态复位 busy/done/errDone;
*)
METHOD Act_Init_Status
VAR_INPUT
END_VAR
actStep.Act_Init();
END_METHOD

METHOD PRIVATE ActionRun
VAR_INPUT
	tempActStep:ITFActStep;
END_VAR
VAR
END_VAR
VAR_STAT//此处定义静态变量, 保证每次进入该函数时能够在线监控当前值
	tempStep:DINT;
END_VAR
tempStep:=tempActStep.getStep();
CASE tempStep OF
0:
	IF tempActStep.isEx() THEN
		tempActStep.setBusyFlag();
		tempActStep.toBeginStep();
	END_IF
	t1(IN:= FALSE );
	t2(IN:= FALSE );
	t3(IN:= FALSE );
10:
	gShowLogTextTitle:='Load Lock Vent';
	IF gRunningState<>RunningStatus.eErrorState THEN
		tempActStep.addStep(10,FALSE);
	ELSE
		error_Trigger(105);
		IF gCtrlMode=ControlMode.eManualCtrMode THEN
			tempActStep.toErrDoneStep();
		END_IF
	END_IF
20:
	IF NOT gICP.ForeLineGauge.error AND gICP.ForeLineGauge.outputValue<gRoughtPumVaccum*10 THEN
		tempActStep.addStep(10,FALSE);
	ELSE
		error_Trigger(107);
		IF gCtrlMode=ControlMode.eManualCtrMode THEN
			tempActStep.toErrDoneStep();
		END_IF
	END_IF
30:
	IF NOT gICP.LoadLockGauge.error AND gICP.LoadLockGauge.outputValue>gATMPressure THEN
		tempActStep.toDoneStep();
	ELSE
		error_Trigger(107);
		tempActStep.addStep(10,FALSE);
	END_IF
40:
	IF gICP.ForlinLineValveExtRelay THEN
		forelineOpenflag:=TRUE;
	ELSE
		forelineOpenflag:=FALSE;
	END_IF
	IF gICP.PDVOpenSensor THEN
		pdvOpenflag:=TRUE;
	ELSE
		pdvOpenflag:=FALSE;
	END_IF
	tempActStep.toStep(100,FALSE);
100:
	tempActStep.addStep(10,TRUE);
110:
	IF NOT gRoughRemain THEN
		S_RoughPumping.Act_Init_Status();
		S_RoughPumping.Act_Ex();
		tempActStep.addStep(10,FALSE);
	ELSE
		tempActStep.toStep(160,FALSE);
	END_IF
120:
	IF S_RoughPumping.done THEN
		gShowLogTextTitle:='Load Lock Pumping';
		tempActStep.addStep(10,FALSE);
	END_IF
	IF S_RoughPumping.errDone THEN
		tempActStep.toStep(100,FALSE);
	END_IF
130:
	tempActStep.addStep(10,FALSE);
140:
	IF gICP.ForlinLineValve.Act_Retract() AND gICP.PDV.Act_Retract() THEN
		gRunningLog.append(CONCAT('LL Vent POU Run:',DINT_TO_STRING(tempStep)));
		gRunningLog.append('LL Vent POU Run:ForLineValve And PDV Close');
		tempActStep.addStep(10,FALSE);
	END_IF
150:
	IF gICP.ForlinLineValve.Get_Done_Ret() AND gICP.PDV.Get_Done_Ret() AND gICP.PDVCloseSensor THEN
		tempActStep.toStep(200,FALSE);
		gRunningLog.append(CONCAT('LL Vent POU Run:',DINT_TO_STRING(tempStep)));
		gRunningLog.append('LL Vent POU Run:ForLineValve And PDV Close Done');
	END_IF
160:
	S_ActuatorRecoveryPOU.Act_Init_Status();
	S_ActuatorRecoveryPOU.Act_Ex();
	tempActStep.addStep(10,FALSE);
170:
	IF S_ActuatorRecoveryPOU.done THEN
		tempActStep.addStep(10,FALSE);
	END_IF
180:
	tempActStep.addStep(10,FALSE);
190:
	tempActStep.addStep(10,FALSE);
200:
	tempActStep.addStep(10,TRUE);
210:
	IF gICP.GateDoorValve.Get_Done_Ret() AND gICP.GateDoorRetSensor AND
		gICP.VentValve.Get_Done_Ret() AND NOT gICP.VentExtRelay AND
		gICP.SlowPummingValve.Get_Done_Ret() AND NOT gICP.SlowPummingExtRelay AND
		gICP.FastPummingValve.Get_Done_Ret() AND NOT gICP.FastPummingExtRelay AND
		gICP.ForlinLineValve.Get_Done_Ret() AND NOT gICP.ForlinLineValveExtRelay AND
		gICP.RoughValve.Get_Done_Ret() AND NOT gICP.RoughValveExtRelay  THEN
		tempActStep.addStep(10,FALSE);		
	END_IF
220:
	IF gICP.VentValve.Act_Extend() THEN
		gRunningLog.append(CONCAT('LL Vent POU Run:',DINT_TO_STRING(tempStep)));
		gRunningLog.append('LL Vent POU Run: Vent Valve Open');
		tempActStep.addStep(10,FALSE);
	END_IF
230:
	IF gICP.VentValve.Get_Done_Ext() THEN
		gRunningLog.append(CONCAT('LL Vent POU Run:',DINT_TO_STRING(tempStep)));
		gRunningLog.append('LL Vent POU Run: Vent Valve Open Done');
		tempActStep.addStep(10,FALSE);
	END_IF
240:
	t2(IN:= gICP.LoadLockGauge.outputValue>gATMPressure,PT:=T#25S );
	IF t2.Q OR NOT gICP.I_LLSwitch THEN
		t1(IN:= FALSE );
		t2(IN:= FALSE );
		t3(IN:= FALSE );
		gRunningLog.append(CONCAT('LL Vent POU Run:',DINT_TO_STRING(tempStep)));
		gRunningLog.append(CONCAT('LL Vent POU Run:LL Vent Pressure Arrive：',REAL_TO_STRING(gICP.LoadLockGauge.outputValue)));
		tempActStep.addStep(10,FALSE);
		RETURN;
	END_IF
	t1(IN:= TRUE,PT:=timeOutTime );
	IF t1.Q THEN
		t1(IN:= FALSE );
		t2(IN:= FALSE );
		t3(IN:= FALSE );
		error_Trigger(109);
		tempActStep.toStep(200,FALSE);
		RETURN;
	END_IF
250:
	tempActStep.addStep(10,TRUE);
260:
	IF gICP.VentValve.Act_Retract() THEN
		gRunningLog.append(CONCAT('LL Vent POU Run:',DINT_TO_STRING(tempStep)));
		gRunningLog.append('LL Vent POU Run: Vent Valve Close');
		tempActStep.addStep(10,FALSE);
	END_IF
270:
	IF gICP.VentValve.Get_Done_Ret() THEN
		gRunningLog.append(CONCAT('LL Vent POU Run:',DINT_TO_STRING(tempStep)));
		gRunningLog.append('LL Vent POU Run: Vent Valve Close Done');
		tempActStep.addStep(10,FALSE);
	END_IF
280:
	t3(IN:=TRUE,PT:=T#1S);
	IF t3.Q THEN
		t1(IN:= FALSE );
		t2(IN:= FALSE );
		t3(IN:= FALSE );
		tempActStep.addStep(10,FALSE);
	END_IF
290:
	tempActStep.toStep(370,FALSE);
370:
	tempActStep.addStep(10,TRUE);
380:
	IF forelineOpenflag THEN
		IF gICP.ForlinLineValve.Act_Extend() THEN
			gRunningLog.append(CONCAT('LL Vent POU Run:',DINT_TO_STRING(tempStep)));
			gRunningLog.append('LL Vent POU Run: ForLine Valve Open ');
			tempActStep.addStep(10,FALSE);
		END_IF
	ELSE
		tempActStep.addStep(20,FALSE);
	END_IF
390:
	IF gICP.ForlinLineValve.Get_Done_Ext() THEN
		gRunningLog.append(CONCAT('LL Vent POU Run:',DINT_TO_STRING(tempStep)));
		gRunningLog.append('LL Vent POU Run: ForLine Valve Open Done');
		tempActStep.addStep(10,FALSE);
	END_IF
400:
	tempActStep.addStep(10,TRUE);
//465:
//	IF gICP.PDV.Act_ChangePos() THEN
//		tempActStep.addStep(2,FALSE);
//	END_IF
//467:
//	IF gICP.PDV.PosMode THEN
//		tempActStep.addStep(3,FALSE);
//	END_IF
410:
	IF pdvOpenflag THEN
		IF gICP.PDV.Act_Open() THEN
			gRunningLog.append(CONCAT('LL Vent POU Run:',DINT_TO_STRING(tempStep)));
			gRunningLog.append('LL Vent POU Run: PDV Open ');
			tempActStep.addStep(10,FALSE);
		END_IF
	ELSE
		tempActStep.toStep(1000,FALSE);
	END_IF
420:
	IF gICP.PDV.Get_Done_Ext() OR gICP.PDVOpenSensor THEN
		gRunningLog.append(CONCAT('LL Vent POU Run:',DINT_TO_STRING(tempStep)));
		gRunningLog.append('LL Vent POU Run: PDV Open Done');
		tempActStep.addStep(10,FALSE);
	END_IF
430:
	tempActStep.toStep(1000,FALSE);
1000:
	tempActStep.toDoneStep();

60000://Done
	tempActStep.setDoneFlag();
	tempActStep.toZeroStep();
	
65000://Error
	tempActStep.setErrDoneFlag();
	tempActStep.toZeroStep();
	gICP.VentValve.Act_Retract();
END_CASE
END_METHOD

END_PROGRAM

// ---- POUs/MachinePOU/SemiAutomatic/S_MachinePumping.TcPOU
PROGRAM S_MachinePumping
VAR_INPUT
	bInit				:BOOL:=FALSE;// 初始化状态 busy/done/errDone
	bTrig				:BOOL:=FALSE;// 执行触发 信号
	bReset				:BOOL:=FALSE;// 报错 复位
	bPause				:BOOL:=FALSE;// 暂停 运行
	bStop				:BOOL:=FALSE;// 停止 运行
	bAbort				:BOOL:=FALSE;// 中止 运行
	
END_VAR
VAR_OUTPUT
	busy				:BOOL;
	done				:BOOL;
	errDone				:BOOL;
END_VAR
VAR
	actStep				:ActStepBase;
END_VAR
VAR
	i: INT;
	t1:ton;
	t2:ton;
	t3:ton;
	notchoose:BOOL;
	timeOutTime:TIME:=T#120S;
	safecheckTime:TIME:=T#1S;
END_VAR

busy:=actStep.isBusy();
done:=actStep.isDone();
errDone:=actStep.isError();
actStep.Act_Pause(pause:=bPause);

IF bTrig THEN
	bTrig:=FALSE;
	IF NOT busy THEN
		actStep.Act_ex();
	END_IF
END_IF

//状态复位
IF bInit THEN
	bInit:=FALSE;
	Act_init_status();
END_IF

IF bAbort OR bStop THEN
	bAbort:=FALSE;
	bStop:=FALSE;
	Act_init_status();
	actStep.toZeroStep();
	gShowLogTextTitle:='NON';
END_IF
ActionRun(tempActStep:=actStep);

(*
---Trigger action
*)
METHOD Act_Ex : BOOL
VAR_INPUT
END_VAR
IF NOT busy THEN
	actStep.Act_ex();
	Act_Ex:=TRUE;
ELSE
	Act_Ex:=FALSE;
END_IF
END_METHOD

(*
---功能: 状态复位 busy/done/errDone;
*)
METHOD Act_Init_Status
VAR_INPUT
END_VAR
actStep.Act_Init();
END_METHOD

METHOD PRIVATE ActionRun
VAR_INPUT
	tempActStep:ITFActStep;
END_VAR
VAR
END_VAR
VAR_STAT//此处定义静态变量, 保证每次进入该函数时能够在线监控当前值
	tempStep:DINT;
END_VAR
tempStep:=tempActStep.getStep();
CASE tempStep OF
0:
	IF tempActStep.isEx() THEN
		tempActStep.setBusyFlag();
		tempActStep.toBeginStep();
	END_IF
	t1(IN:= FALSE );
	t2(IN:= FALSE );
	t3(IN:= FALSE );
10:
	gShowLogTextTitle:='Machine Pumping';
	IF gRunningState<>RunningStatus.eErrorState THEN
		tempActStep.addStep(10,FALSE);
	ELSE
		error_Trigger(105);
		tempActStep.toErrDoneStep();
	END_IF
20:
	IF NOT gICP.ForeLineGauge.error AND gICP.ForeLineGauge.outputValue<gRoughtPumVaccum*10 THEN
		tempActStep.addStep(10,FALSE);
	ELSE
		error_Trigger(107);
		tempActStep.toErrDoneStep();
	END_IF
30:
	tempActStep.toStep(200,FALSE);
200:
	tempActStep.addStep(10,TRUE);
210:
	S_RoughPumping.Act_Init_Status();
	S_RoughPumping.Act_Ex();
	tempActStep.addStep(10,FALSE);
220:
	IF S_RoughPumping.done THEN
		gShowLogTextTitle:='Machine Pumping';
		ups_CX51X0.Act_Wrtie();
		tempActStep.addStep(10,FALSE);
	END_IF
	IF S_RoughPumping.errDone THEN
		tempActStep.toErrDoneStep();
	END_IF
230:
	tempActStep.toStep(1000,FALSE);
1000:
	tempActStep.toDoneStep();

60000://Done
	tempActStep.setDoneFlag();
	tempActStep.toZeroStep();
	
65000://Error
	tempActStep.setErrDoneFlag();
	tempActStep.toZeroStep();
END_CASE
END_METHOD

END_PROGRAM

// ---- POUs/MachinePOU/SemiAutomatic/S_WaferCheckPOU.TcPOU
PROGRAM S_WaferCheckPOU
VAR_INPUT
	bInit				:BOOL:=FALSE;// 初始化状态 busy/done/errDone
	bTrig				:BOOL:=FALSE;// 执行触发 信号
	bReset				:BOOL:=FALSE;// 报错 复位
	bPause				:BOOL:=FALSE;// 暂停 运行
	bStop				:BOOL:=FALSE;// 停止 运行
	bAbort				:BOOL:=FALSE;// 中止 运行
	
END_VAR
VAR_OUTPUT
	busy				:BOOL;
	done				:BOOL;
	errDone				:BOOL;
END_VAR
VAR
	actStep				:ActStepBase;
END_VAR
VAR
	i: INT;
	t1:ton;
	t2:ton;
	t3:ton;
	notchoose:BOOL;
	timeOutTime:TIME:= T#60S;
END_VAR

busy:=actStep.isBusy();
done:=actStep.isDone();
errDone:=actStep.isError();
actStep.Act_Pause(pause:=bPause);

IF bTrig THEN
	bTrig:=FALSE;
	IF NOT busy THEN
		gShowLogTextTitle:='Wafer Check';
		actStep.Act_ex();
	END_IF
END_IF

//状态复位
IF bInit THEN
	bInit:=FALSE;
	Act_init_status();
END_IF

IF bAbort OR bStop THEN
	bAbort:=FALSE;
	bStop:=FALSE;
	Act_init_status();
	actStep.toZeroStep();
	gShowLogTextTitle:='NON';
END_IF
ActionRun(tempActStep:=actStep);

(*
---Trigger action
*)
METHOD Act_Ex : BOOL
VAR_INPUT
END_VAR
IF NOT busy THEN
	actStep.Act_ex();
	Act_Ex:=TRUE;
ELSE
	Act_Ex:=FALSE;
END_IF
END_METHOD

(*
---功能: 状态复位 busy/done/errDone;
*)
METHOD Act_Init_Status
VAR_INPUT
END_VAR
actStep.Act_Init();
END_METHOD

METHOD PRIVATE ActionRun
VAR_INPUT
	tempActStep:ITFActStep;
END_VAR
VAR
END_VAR
VAR_STAT//此处定义静态变量, 保证每次进入该函数时能够在线监控当前值
	tempStep:DINT;
END_VAR
tempStep:=tempActStep.getStep();
CASE tempStep OF
0:
	IF tempActStep.isEx() THEN
		tempActStep.setBusyFlag();
		tempActStep.toBeginStep();
	END_IF
	t1(IN:= FALSE );
	t2(IN:= FALSE );
	t3(IN:= FALSE );
10:
	IF gRunningState<>RunningStatus.eErrorState THEN
		tempActStep.addStep(10,FALSE);
	ELSE
		tempActStep.toErrDoneStep();
	END_IF
20:
	gEnableWaferCheck:=2;
	tempActStep.addStep(10,FALSE);
30:
	IF gEnableWaferCheck=0 THEN// 不检测直接完成
		tempActStep.toStep(100,FALSE);
		t1(IN:= FALSE );
		t2(IN:= FALSE );
		t3(IN:= FALSE );
		RETURN;
	END_IF
	IF gEnableWaferCheck=1 THEN// 检测逻辑
		t1(IN:= FALSE );
		t2(IN:= FALSE );
		t3(IN:= FALSE );
		tempActStep.toStep(100,FALSE);
		RETURN;
	END_IF
	t3(IN:=TRUE,PT:=timeOutTime);
	IF t3.Q THEN
		t1(IN:= FALSE );
		t2(IN:= FALSE );
		t3(IN:= FALSE );
		tempActStep.toErrDoneStep();
		RETURN;
	END_IF
100:
	IF NOT gICP.I_WaferCheck THEN
		tempActStep.addStep(10,FALSE);
	ELSE
		// 机械臂上有晶圆，又需要进行晶圆检测，直接报错
		tempActStep.toErrDoneStep();
	END_IF
110:
	tempActStep.addStep(10,TRUE);
120:
	S_RoughPumping.Act_Init_Status();
	S_RoughPumping.Act_Ex();
	tempActStep.addStep(10,FALSE);
130:
	IF S_RoughPumping.done THEN
		tempActStep.addStep(5,FALSE);
	END_IF
	IF S_RoughPumping.errDone THEN
		tempActStep.toErrDoneStep();
	END_IF	
135:
	IF gEnableWaferCheck=0 THEN// 不检测直接完成
		tempActStep.toDoneStep();
		t1(IN:= FALSE );
		t2(IN:= FALSE );
		t3(IN:= FALSE );
		RETURN;
	END_IF
	IF gEnableWaferCheck=1 THEN// 检测逻辑
		t1(IN:= FALSE );
		t2(IN:= FALSE );
		t3(IN:= FALSE );
		tempActStep.addStep(5,FALSE);
		RETURN;
	END_IF
140:
	IF gICP.PDV.Act_Retract() THEN
		tempActStep.addStep(10,FALSE);
	END_IF
150:
	IF gICP.PDV.Get_Done_Ret() OR gICP.PDVCloseSensor THEN
		tempActStep.addStep(10,FALSE);
	END_IF
160:
	tempActStep.addStep(10,TRUE);
170:
	IF gICP.GateDoorValve.Act_Extend() THEN
		tempActStep.addStep(10,FALSE);
	END_IF
180:
	IF gICP.GateDoorValve.Get_Done_Ext() AND gICP.GateDoorExtSensor THEN
		tempActStep.addStep(10,FALSE);
	END_IF
190:
	tempActStep.addStep(10,TRUE);
200:
	IF NOT gICP.ElectrodeCylRetSensor THEN
		tempActStep.addStep(10,FALSE);
	ELSE
		tempActStep.addStep(30,FALSE);
	END_IF
210:
	tempActStep.addStep(10,TRUE);
220:
	IF gICP.ElectrodeCyl.Act_Retract() THEN
		tempActStep.addStep(10,FALSE);
	END_IF
230:
	IF gICP.ElectrodeCyl.Get_Done_Ret() AND gICP.ElectrodeCylRetSensor THEN
		tempActStep.addStep(10,FALSE);
	END_IF
240:
	tempActStep.addStep(10,TRUE);
250:
	IF gICP.LiftPinCyl.Act_Extend() THEN
		tempActStep.addStep(10,FALSE);
	END_IF
260:
	IF gICP.LiftPinCyl.Get_Done_Ext() AND gICP.LiftPinExtSensor THEN
		tempActStep.addStep(10,FALSE);
	END_IF
270:
	tempActStep.addStep(10,TRUE);
280:
	IF gICP.ARM.Act_HOME_Auto() THEN
		tempActStep.addStep(10,FALSE);
	END_IF
290:
	IF NOT gICP.I_ARMHome THEN// 手臂当前不应该在原点位置
		tempActStep.addStep(10,FALSE);
	END_IF
300:
	t2(IN:=TRUE,PT:=T#10S);
	IF t2.Q AND gICP.ARM.Get_Done_IN() THEN
		t1(IN:= FALSE );
		t2(IN:= FALSE );
		t3(IN:= FALSE );
		tempActStep.toErrDoneStep();
		RETURN;
	END_IF
310:
	tempActStep.addStep(10,TRUE);
320:
	IF gICP.LiftPinCyl.Act_Retract() THEN
		tempActStep.addStep(10,FALSE);
	END_IF
330:
	IF gICP.LiftPinCyl.Get_Done_Ret() AND gICP.LiftPinRetSensor THEN
		tempActStep.addStep(10,FALSE);
	END_IF
340:
	tempActStep.addStep(10,TRUE);
350:
	IF gICP.ARM.Act_HOME_Auto() THEN
		tempActStep.addStep(10,FALSE);
	END_IF
360:
	IF gICP.ARM.Get_Done_HOME() AND gICP.I_ARMHome THEN// 手臂当前不应该在原点位置
		tempActStep.addStep(10,FALSE);
	END_IF
370:
	t2(IN:=TRUE,PT:=T#1S);
	IF t2.Q THEN
		t1(IN:= FALSE );
		t2(IN:= FALSE );
		t3(IN:= FALSE );
		tempActStep.toErrDoneStep();
		RETURN;
	END_IF
380:
	tempActStep.addStep(10,TRUE);
390:
	IF gICP.GateDoorValve.Act_Retract() THEN
		tempActStep.addStep(10,FALSE);
	END_IF
400:
	IF gICP.GateDoorValve.Get_Done_Ret() AND gICP.GateDoorRetSensor THEN
		tempActStep.addStep(10,FALSE);
	END_IF
410:
	IF gICP.I_WaferCheck THEN
		;// wafer记忆状态更新
	ELSE
		;// wafer记忆状态更新
	END_IF
	tempActStep.addStep(10,FALSE);
420:
	tempActStep.toDoneStep();
1000:
	tempActStep.toDoneStep();

60000://Done
	tempActStep.setDoneFlag();
	tempActStep.toZeroStep();
	
65000://Error
	tempActStep.setErrDoneFlag();
	tempActStep.toZeroStep();
END_CASE
END_METHOD

END_PROGRAM

// ---- POUs/MachinePOU/SemiAutomatic/S_PDVSafeCtr.TcPOU
PROGRAM S_PDVSafeCtr
VAR_INPUT
	bInit				:BOOL:=FALSE;// 初始化状态 busy/done/errDone
	bTrig				:BOOL:=FALSE;// 执行触发 信号
	bReset				:BOOL:=FALSE;// 报错 复位
	bPause				:BOOL:=FALSE;// 暂停 运行
	bStop				:BOOL:=FALSE;// 停止 运行
	bAbort				:BOOL:=FALSE;// 中止 运行
	
END_VAR
VAR_OUTPUT
	busy				:BOOL;
	done				:BOOL;
	errDone				:BOOL;
	stopDone			:BOOL;
END_VAR
VAR
	actStep				:ActStepBase;
END_VAR
VAR
	i: INT;
	t1:ton;
	t2:ton;
	t3:ton;
	openErrorDelayTon:TON;
	notchoose:BOOL;
	timeOutTime:TIME:= T#60S;
	ventTime:TIME:=T#15S;
	chamberVaccum:REAL;
	TBVaccum:REAL;
	vaccumAbs:REAL:=500;
	ATMVaccum:REAL:=200000;
	forlineOpen:BOOL;
	roughtOpen:BOOL;
	rtrig:R_TRIG;
END_VAR

busy:=actStep.isBusy();
done:=actStep.isDone();
errDone:=actStep.isError();
actStep.Act_Pause(pause:=bPause);
rtrig(CLK:=gPDVOpencondition);
IF bTrig OR rtrig.Q THEN
	bTrig:=FALSE;
	Act_init_status();
	IF NOT busy THEN
		actStep.Act_ex();
	END_IF
END_IF

//状态复位
IF bInit THEN
	bInit:=FALSE;
	Act_init_status();
END_IF

IF bAbort OR bStop THEN
	bAbort:=FALSE;
	bStop:=FALSE;
	Act_init_status();
	actStep.toZeroStep();
	IF gPDVOpencondition THEN
		gPDVOpencondition:=FALSE;
		gICP.PDV.Act_Retract();
		IF NOT forlineOpen THEN
			gICP.ForlinLineValve.Act_Retract();
		END_IF
		IF forlineOpen THEN
			gICP.ForlinLineValve.Act_Extend();
		END_IF
		IF NOT roughtOpen THEN
			gICP.RoughValve.Act_Retract();
		END_IF
		IF roughtOpen THEN
			gICP.RoughValve.Act_Extend();
		END_IF
	END_IF
END_IF
ActionRun(tempActStep:=actStep);

(*
---Trigger action
*)
METHOD Act_Ex : BOOL
VAR_INPUT
END_VAR
IF NOT busy THEN
	actStep.Act_ex();
	Act_Ex:=TRUE;
ELSE
	Act_Ex:=FALSE;
END_IF
END_METHOD

(*
---功能: 状态复位 busy/done/errDone;
*)
METHOD Act_Init_Status
VAR_INPUT
END_VAR
actStep.Act_Init();
END_METHOD

METHOD PRIVATE ActionRun
VAR_INPUT
	tempActStep:ITFActStep;
END_VAR
VAR_STAT//此处定义静态变量, 保证每次进入该函数时能够在线监控当前值
	tempStep:DINT;
END_VAR
tempStep:=tempActStep.getStep();
CASE tempStep OF
0:
	IF tempActStep.isEx() THEN
		tempActStep.setBusyFlag();
		tempActStep.toBeginStep();
	END_IF
	t1(IN:= FALSE );
	t2(IN:= FALSE );
	t3(IN:= FALSE );
10:
	IF (gICP.TruboPumOpen AND gICP.TruboPumNormal) OR (NOT gICP.TruboPumOpen AND gICP.TruboPumNoRotation) THEN
		IF gICP.ForlinLineValveExtRelay THEN
			forlineOpen:=TRUE;
		ELSE
			forlineOpen:=FALSE;
		END_IF
		IF gICP.RoughValveExtRelay THEN
			roughtOpen:=TRUE;
		ELSE
			roughtOpen:=FALSE;
		END_IF
		IF gPDVOpencondition THEN
			gRunningLog.append(CONCAT('PDV Open Safety Check:',DINT_TO_STRING(tempStep)));
			gRunningLog.append('PDV Open Safety Check:Differential Pressure Check');
			tempActStep.addStep(10,FALSE);
		END_IF
	ELSE
		error_Trigger(103);
		tempActStep.toErrDoneStep();
	END_IF
20:
	IF gICP.RoughValve.Act_Retract() AND gICP.ForlinLineValve.Act_Retract() AND gICP.FastPummingValve.Act_Retract() AND gICP.SlowPummingValve.Act_Retract() THEN
		gRunningLog.append(CONCAT('PDV Open Safety Check:',DINT_TO_STRING(tempStep)));
		gRunningLog.append('PDV Open Safety Check:RoughValve | ForeLineValve | FastPuming | SlowPuming Close');
		tempActStep.addStep(10,FALSE);
	END_IF
30:
	t1(IN:= TRUE,PT:=T#1S );
	IF t1.Q THEN
		t1(IN:= FALSE );
		t2(IN:= FALSE );
		t3(IN:= FALSE );
		tempActStep.addStep(10,FALSE);
	END_IF
40:
	IF gICP.RoughValve.Get_Done_Ret() AND gICP.ForlinLineValve.Get_Done_Ret() AND gICP.FastPummingValve.Get_Done_Ret() AND gICP.SlowPummingValve.Get_Done_Ret() THEN
		gRunningLog.append(CONCAT('PDV Open Safety Check:',DINT_TO_STRING(tempStep)));
		gRunningLog.append('PDV Open Safety Check:RoughValve | ForeLineValve | FastPuming | SlowPuming Close Done');
		tempActStep.addStep(10,FALSE);
	END_IF
50:
	t2(IN:= TRUE,PT:=T#1S );
	IF t2.Q THEN
		t1(IN:= FALSE );
		t2(IN:= FALSE );
		t3(IN:= FALSE );
		tempActStep.addStep(10,FALSE);
	END_IF
60:
	IF gICP.RoughValve.Act_Extend() THEN
		gRunningLog.append(CONCAT('PDV Open Safety Check:',DINT_TO_STRING(tempStep)));
		gRunningLog.append('PDV Open Safety Check:RoughValve Open');
		tempActStep.addStep(10,FALSE);
	END_IF
70:
	t3(IN:= TRUE,PT:=T#1S );
	IF t3.Q AND gICP.RoughValve.Get_Done_Ext() THEN
		t1(IN:= FALSE );
		t2(IN:= FALSE );
		t3(IN:= FALSE );
		tempActStep.addStep(10,FALSE);
		gRunningLog.append(CONCAT('PDV Open Safety Check:',DINT_TO_STRING(tempStep)));
		gRunningLog.append('PDV Open Safety Check:RoughValve Open');
		chamberVaccum:=gICP.ForeLineGauge.outputValue;
		gICP.RoughValve.Act_Retract();
	END_IF
80:
	IF gICP.RoughValve.Get_Done_Ret() THEN
		gRunningLog.append(CONCAT('PDV Open Safety Check:',DINT_TO_STRING(tempStep)));
		gRunningLog.append('PDV Open Safety Check:RoughValve Open Done');
		tempActStep.addStep(5,FALSE);
	END_IF
85:
	t3(IN:= TRUE,PT:=T#10S );
	IF t3.Q AND gICP.RoughValve.Get_Done_Ret() AND gICP.ForeLineGauge.outputValue<gRoughtPumVaccum THEN
		gRunningLog.append(CONCAT('PDV Open Safety Check:',DINT_TO_STRING(tempStep)));
		gRunningLog.append(CONCAT('PDV Open Safety Check:ForeLine Gauge Pressure Arrive: ',REAL_TO_STRING(gICP.ForeLineGauge.outputValue)));
		t1(IN:= FALSE );
		t2(IN:= FALSE );
		t3(IN:= FALSE );
		tempActStep.addStep(2,FALSE);
	END_IF
87:
	t2(IN:= TRUE,PT:=T#3S );
	IF t2.Q THEN
		t1(IN:= FALSE );
		t2(IN:= FALSE );
		t3(IN:= FALSE );
		tempActStep.addStep(3,FALSE);
	END_IF
90:
	IF gICP.ForlinLineValve.Act_Extend() THEN
		gRunningLog.append(CONCAT('PDV Open Safety Check:',DINT_TO_STRING(tempStep)));
		gRunningLog.append('PDV Open Safety Check:ForLineValve Open');
		tempActStep.addStep(10,FALSE);
	END_IF
100:
	t3(IN:= TRUE,PT:=T#1S );
	IF t3.Q AND gICP.ForlinLineValve.Get_Done_Ext() THEN
		t1(IN:= FALSE );
		t2(IN:= FALSE );
		t3(IN:= FALSE );
		tempActStep.addStep(5,FALSE);
		gRunningLog.append(CONCAT('PDV Open Safety Check:',DINT_TO_STRING(tempStep)));
		gRunningLog.append('PDV Open Safety Check:ForLineValve Open Done and Remain Foreline Gauge Pressure');
		TBVaccum:=gICP.ForeLineGauge.outputValue;
	END_IF
105:
	IF gICP.ForlinLineValve.Act_Retract() THEN
		gRunningLog.append(CONCAT('PDV Open Safety Check:',DINT_TO_STRING(tempStep)));
		gRunningLog.append('PDV Open Safety Check:ForLineValve Close');
	END_IF
110:
	IF gICP.ForlinLineValve.Get_Done_Ret() THEN
		gRunningLog.append(CONCAT('PDV Open Safety Check:',DINT_TO_STRING(tempStep)));
		gRunningLog.append('PDV Open Safety Check:ForLineValve Close Done');
		tempActStep.addStep(10,FALSE);
	END_IF
120:
	IF ( TBVaccum>ATMVaccum AND chamberVaccum>ATMVaccum ) OR ABS(TBVaccum-chamberVaccum)<vaccumAbs THEN
		tempActStep.addStep(10,FALSE);
		gPDVOpencondition:=FALSE;
		gRunningLog.append(CONCAT('PDV Open Safety Check:',DINT_TO_STRING(tempStep)));
		gRunningLog.append('PDV Open Safety Check:PDV Open');
	ELSE
		error_Trigger(104);
		tempActStep.toErrDoneStep();
	END_IF
130:
	IF (gICP.PDV.Get_Done_Ext() OR gICP.PDVOpenSensor) THEN
		IF forlineOpen AND NOT roughtOpen THEN
			tempActStep.addStep(10,FALSE);
			RETURN;
		END_IF
		IF NOT forlineOpen AND roughtOpen THEN
			tempActStep.addStep(160,FALSE);
			RETURN;
		END_IF
		IF NOT forlineOpen AND NOT roughtOpen THEN
			tempActStep.toStep(1000,FALSE);
			RETURN;
		END_IF
	END_IF
140:
	IF gICP.ForlinLineValve.Act_Extend() THEN
		gRunningLog.append(CONCAT('PDV Open Safety Check:',DINT_TO_STRING(tempStep)));
		gRunningLog.append('PDV Open Safety Check:ForLineValve Open');
		tempActStep.addStep(10,FALSE);
	END_IF
150:
	IF gICP.ForlinLineValve.Get_Done_Ext() THEN
		gRunningLog.append(CONCAT('PDV Open Safety Check:',DINT_TO_STRING(tempStep)));
		gRunningLog.append('PDV Open Safety Check:ForLineValve Open Done');
		tempActStep.addStep(10,FALSE);
	END_IF
160:
	tempActStep.toStep(1000,FALSE);
200:
	IF gICP.RoughValve.Act_Extend() THEN
		gRunningLog.append(CONCAT('PDV Open Safety Check:',DINT_TO_STRING(tempStep)));
		gRunningLog.append('PDV Open Safety Check:RoughValve Open');
		tempActStep.addStep(10,FALSE);
	END_IF
210:
	IF gICP.RoughValve.Get_Done_Ext() THEN
		gRunningLog.append(CONCAT('PDV Open Safety Check:',DINT_TO_STRING(tempStep)));
		gRunningLog.append('PDV Open Safety Check:RoughValve Open Done');
		tempActStep.addStep(10,FALSE);
	END_IF
220:
	gRunningLog.append('PDV Open Safety Check:Differential Pressure Check Done');
	tempActStep.toStep(1000,FALSE);
1000:
	tempActStep.toDoneStep();
60000://Done
	tempActStep.setDoneFlag();
	tempActStep.toZeroStep();
65000://Error
	tempActStep.setErrDoneFlag();
	tempActStep.toZeroStep();
	gICP.PDV.Act_Retract();
	gPDVOpencondition:=FALSE;
	gICP.RoughValve.Act_Retract();
	gICP.ForlinLineValve.Act_Retract();
	gICP.FastPummingValve.Act_Retract();
	gICP.SlowPummingValve.Act_Retract();
END_CASE
END_METHOD

END_PROGRAM

// ---- POUs/Communication/PRG_ADS_Comm_ByName_A2B.TcPOU
PROGRAM PRG_ADS_Comm_ByName_A2B
VAR
	// 1808ErrorID 多数是ADS访问变量出错，需要仔细查看变量名称是否有误
	fbGetHandle					: ADSRDWRT;				//获取句柄功能块
	fbADSGetData				: ADSREAD;				//A机从B机读功能块
	fbADSSendData				: ADSWRITE;				//A机向B机写功能块
	iHandle_A_R					: UDINT			:= 0;	//A机接收数据句柄
	iHandle_A_T					: UDINT			:= 0;	//A机向B机写收据句柄
	sVarName					:STRING;				//结构体变量名
	AdsNETID					: T_AmsNetId	:= '5.117.124.188.1.1';//B机AMS Net Id   ICP:5.114.113.208.1.1
	AdsPort						:T_AmsPort		:=851;	//B机PLC端口号
	iADSCommStep				:INT;
	iDelayTM					:INT;
	bAdsCommErr					:BOOL;
	tHeartBeat					:TON;
	tON							:TON;
	tOFF						:TON;
END_VAR

MsgMap_A2B();
CASE iADSCommStep OF
0:// 获取gSTA2BData句柄-----TC3定义全局变量，必须加'GVL.'.-----ADSIGRP_SYM_HNDBYNAME----A---->Write to---->C
	sVarName					:='GVL_AllGLOBAL.gSTA2BData';
	fbGetHandle(NETID:=AdsNETID , PORT:=AdsPort , IDXGRP:=ADSIGRP_SYM_HNDBYNAME , IDXOFFS:=16#00 , WRITELEN:=INT_TO_UDINT(len(sVarName)) ,
	 READLEN:=SIZEOF(iHandle_A_T) , SRCADDR:=ADR(sVarName) , DESTADDR:=ADR(iHandle_A_T) , WRTRD:= FALSE, );
	IF iDelayTM>200 THEN
		iDelayTM				:=0;
		iADSCommStep			:=iADSCommStep+1;
	ELSE
		iDelayTM				:=iDelayTM+1;
	END_IF
1:
	IF NOT fbGetHandle.BUSY THEN
		iADSCommStep			:=iADSCommStep+1;
	ELSE
		iADSCommStep			:=999;
	END_IF
2:
	fbGetHandle(WRTRD:= TRUE );
	IF fbGetHandle.BUSY THEN
		iADSCommStep			:=iADSCommStep+1;
	ELSE
		iADSCommStep			:=999;
	END_IF
3:
	fbGetHandle(WRTRD:= FALSE );
	IF NOT fbGetHandle.BUSY THEN
		IF NOT fbGetHandle.ERR THEN
			iADSCommStep			:=iADSCommStep+1;
		ELSE
			iADSCommStep			:=999;
		END_IF
	ELSE
		IF iDelayTM>100 THEN
			iDelayTM					:=0;
			iADSCommStep				:=999;
		ELSE
			iDelayTM					:=iDelayTM+1;
		END_IF
	END_IF
4:
	iADSCommStep				:=10;
10://-B---->Write to---->A
	sVarName					:='GVL_AllGLOBAL.gSTB2AData';
	fbGetHandle(NETID:=AdsNETID , PORT:=AdsPort , IDXGRP:=ADSIGRP_SYM_HNDBYNAME , IDXOFFS:=16#00 , WRITELEN:=INT_TO_UDINT(LEN(sVarName)) , 
	READLEN:=SIZEOF(iHandle_A_R) , SRCADDR:=ADR(sVarName) , DESTADDR:=ADR(iHandle_A_R) , WRTRD:= FALSE, );
	iADSCommStep			:=iADSCommStep+1;
11:
	IF NOT fbGetHandle.BUSY THEN
		iADSCommStep			:=iADSCommStep+1;
	ELSE
		iADSCommStep				:=999;
	END_IF
12:
	fbGetHandle(WRTRD:= TRUE );
	IF fbGetHandle.BUSY THEN
		iADSCommStep			:=iADSCommStep+1;
	ELSE
		iADSCommStep				:=999;
	END_IF
13:
	fbGetHandle(WRTRD:= FALSE );
	IF NOT fbGetHandle.BUSY THEN
		IF NOT fbGetHandle.ERR THEN
			iADSCommStep			:=iADSCommStep+1;
		ELSE
			iADSCommStep				:=999;
		END_IF
	ELSE
		IF iDelayTM>100 THEN
			iDelayTM					:=0;
			iADSCommStep				:=999;
		ELSE
			iDelayTM					:=iDelayTM+1;
		END_IF
	END_IF
14:
	iADSCommStep				:=20;
20://'GVL_AllGLOBAL.stA2CData'定义全局变量就这么写。注意-------'IDXGRP:=ADSIGRP_SYM_VALBYHND 'A---->WRITE TO ----C
	fbADSSendData(	NETID:= AdsNETID, PORT:=AdsPort , IDXGRP:=ADSIGRP_SYM_VALBYHND , IDXOFFS:=iHandle_A_T ,
	 LEN:=SIZEOF(GVL_AllGLOBAL.gSTA2BData) , SRCADDR:=ADR(GVL_AllGLOBAL.gSTA2BData) , WRITE:=FALSE ,  );
	iADSCommStep			:=iADSCommStep+1;
21:
	IF 	NOT fbADSSendData.BUSY THEN
		iADSCommStep			:=iADSCommStep+1;
	ELSE
		iADSCommStep				:=999;
	END_IF
22:
	fbADSSendData(WRITE:=TRUE ,);
	IF fbADSSendData.BUSY THEN
		iADSCommStep			:=iADSCommStep+1;
	ELSE
		iADSCommStep				:=999;
	END_IF
23:
	fbADSSendData(WRITE:=FALSE ,);
	IF NOT fbADSSendData.BUSY THEN
		IF NOT  fbADSSendData.ERR THEN
			iADSCommStep			:=iADSCommStep+1;
		ELSE
			iADSCommStep				:=999;
		END_IF
	ELSE
		IF iDelayTM>100 THEN
			iDelayTM					:=0;
			iADSCommStep				:=999;
		ELSE
			iDelayTM					:=iDelayTM+1;
		END_IF
	END_IF
24:
	iADSCommStep			:=30;
30://C---->WRITE TO ----A
	fbADSGetData(NETID:=AdsNETID , PORT:=AdsPort , IDXGRP:=ADSIGRP_SYM_VALBYHND , IDXOFFS:=iHandle_A_R , 
	LEN:=SIZEOF(GVL_AllGLOBAL.gSTB2AData) , DESTADDR:= ADR(GVL_AllGLOBAL.gSTB2AData), READ:=FALSE );
	iADSCommStep				:=iADSCommStep+1;
31:
	IF NOT fbADSGetData.BUSY THEN
		iADSCommStep			:=iADSCommStep+1;
	ELSE
		iADSCommStep			:=999;
	END_IF
32:
	fbADSGetData(READ:=TRUE );
	IF  fbADSGetData.BUSY THEN
		iADSCommStep			:=iADSCommStep+1;
	ELSE
		iADSCommStep			:=999;
	END_IF
33:
	fbADSGetData(READ:=FALSE );
	IF  NOT fbADSGetData.BUSY THEN
		IF NOT fbADSGetData.ERR THEN
			iADSCommStep			:=iADSCommStep+1;
		ELSE
			iADSCommStep				:=999;
		END_IF
	ELSE
		IF iDelayTM>100 THEN
			iDelayTM					:=0;
			iADSCommStep				:=999;
		ELSE
			iDelayTM					:=iDelayTM+1;
		END_IF
	END_IF	
34:
	iADSCommStep			:=20;
999://异常处理
	iADSCommStep			:=0;
END_CASE
//A机建立心跳
tHeartBeat(IN:=NOT tHeartBeat.Q , PT:=T#1S , Q=> , ET=> );
IF tHeartBeat.Q THEN
	gSTA2BData.bHeartBeatMonitor			:=NOT gSTA2BData.bHeartBeatMonitor;
END_IF


// A机监控C机心跳
IF gSTB2AData.bHeartBeatMonitor THEN
	tON(IN:=gSTB2AData.bHeartBeatMonitor , PT:=T#2S , Q=> , ET=> );
	tOFF(IN:=FALSE , PT:=T#2S , Q=> , ET=> );
	IF tON.Q THEN
		bAdsCommErr					:=TRUE;
		gADSConnected				:=FALSE;
	ELSE
		bAdsCommErr					:=FALSE;
		gADSConnected				:=TRUE;
	END_IF
ELSE
	tOFF(IN:=NOT gSTB2AData.bHeartBeatMonitor , PT:=T#2S , Q=> , ET=> );
	tON(IN:=FALSE , PT:=T#2S , Q=> , ET=> );
	IF tOFF.Q THEN
		bAdsCommErr					:=TRUE;
		gADSConnected			:=FALSE;
	ELSE
		bAdsCommErr					:=FALSE;
		gADSConnected			:=TRUE;
	END_IF
END_IF
gSTA2BData.bError:=bAdsCommErr;
MsgMap_B2A();

ACTION MsgClear_AB:
gSTA2BData.Cmd_1:=FALSE;
gSTA2BData.Cmd_2:=FALSE;
gSTA2BData.Cmd_3:=FALSE;
gSTA2BData.Cmd_4:=FALSE;
gSTA2BData.Cmd_5:=FALSE;
gSTA2BData.Cmd_6:=FALSE;
gSTA2BData.Cmd_7:=FALSE;
gSTA2BData.Cmd_8:=FALSE;
gSTA2BData.Cmd_9:=FALSE;
gSTA2BData.Cmd_10:=FALSE;
gSTA2BData.O_1:=FALSE;
gSTA2BData.O_2:=FALSE;
gSTA2BData.O_3:=FALSE;
gSTA2BData.O_4:=FALSE;
gSTA2BData.O_5:=FALSE;
gSTA2BData.O_6:=FALSE;
gSTA2BData.O_7:=FALSE;
gSTA2BData.O_8:=FALSE;
gSTA2BData.O_9:=FALSE;
gSTA2BData.O_10:=FALSE;
END_ACTION

ACTION MsgMap_A2B:
// 变量中转
//gSTA2BData.Cmd_1:=    ;
//gSTA2BData.Cmd_2:=    ;
//gSTA2BData.Cmd_3:=    ;
//gSTA2BData.Cmd_4:=    ;
//gSTA2BData.Cmd_5:=    ;
//gSTA2BData.Cmd_6:=    ;
//gSTA2BData.Cmd_7:=    ;
//gSTA2BData.Cmd_8:=    ;
//gSTA2BData.Cmd_9:=    ;
//gSTA2BData.Cmd_10:=    ;

//gSTA2BData.O_1:=    ;
//gSTA2BData.O_2:=    ;
//gSTA2BData.O_3:=    ;
//gSTA2BData.O_4:=    ;
//gSTA2BData.O_5:=    ;
//gSTA2BData.O_6:=    ;
//gSTA2BData.O_7:=    ;
//gSTA2BData.O_8:=    ;
//gSTA2BData.O_9:=    ;
//gSTA2BData.O_10:=    ;
END_ACTION

ACTION MsgMap_B2A:
// 变量中转
//gSTA2BData.I_1 :=gSTA2BData.I_1     ;
//gSTA2BData.I_2 :=gSTA2BData.I_2     ;
//gSTA2BData.I_3 :=gSTA2BData.I_3     ;
//gSTA2BData.I_4 :=gSTA2BData.I_4     ;
//gSTA2BData.I_5 :=gSTA2BData.I_5     ;
//gSTA2BData.I_6 :=gSTA2BData.I_6     ;
//gSTA2BData.I_7 :=gSTA2BData.I_7     ;
//gSTA2BData.I_8 :=gSTA2BData.I_8     ;
//gSTA2BData.I_9 :=gSTA2BData.I_9     ;
//gSTA2BData.I_10:=gSTA2BData.I_10    ;
END_ACTION

END_PROGRAM

// ---- POUs/BaseModule/Communication/FuncModule_RS232_SRF.TcPOU
PROGRAM FuncModule_RS232_SRF
VAR_INPUT
	serialExcute				:BOOL;// RS232开始一次参数读取
	serialSlaveID				:UINT;// 232从站节点号
	sendstr						:STRING;
	prefix						:STRING:='S';// 字符串头
	suffix						:STRING:= '$R';// 字符串尾
	timeout						:TIME:=T#100MS;// 超时时间
	goPosLoad					:LREAL;
	goPosPhase					:LREAL;
	setPresetExt				:BOOL;
END_VAR
VAR_OUTPUT
	serialBusy						:BOOL;
	setPresetBusy					:BOOL;
	serialDone						:BOOL;
	setPresetDone						:BOOL;
	serialError						:BOOL;
	setPresetError						:BOOL;
	serialConnected					:BOOL;
	load							:REAL;// Load电容
	phase							:REAL;// Phase电容
	rec_ManulOrAuto					:BOOL;// Manul OR Auto
	rec_MAStr						:STRING:='Auto';
	loadRunErr						:BOOL;
	phashRunErr						:BOOL;
END_VAR
VAR
	//Byte方式
	send1:							SendData;
	receive1:						ReceiveString;
 
	Timer1:							TON;
	TimerSetPreset:							TON;
	t1:								TON;
	ITemp:INT;
	arr_SendData:					STRING;(*READ*)//发送数据
	arr_RcvDataString:				STRING;// 接收数据
	arr_RcvDataStringTemp:				STRING;// 接收数据
	arr_RcvDataStringClear:			STRING;// 清除接收数据
	RcvDataFlag:			BOOL;// 接收数据标志位
	serialStep						:UINT;				//处理步数
	serialErrorID					:UINT;
	setPresetStep					:UINT;				//处理步数
	serialTimeOut:BOOL;//接收数据超时
	serialRecError:BOOL;//接收数据错误
	reciveFtrig:F_TRIG;
	recTon:TON;
	againSendS3:TON;
	//字符串方式
	(*send1:							SendString;
	receive1:						ReceiveString;
	
	Timer1:							TON;
	
	_sendString:					STRING:='4567';
	_receive1string:				STRING;
	_recvLast:						STRING;				//保存上一个周期接收的字符*)
	R00_LDMIN:INT:=398;
	R01_LDMAX:INT:=2523;
	R02_PHMIN:INT:=182;
	R03_PHMAX:INT:=3050;
	AD_CH6:INT;
	AD_CH7:INT;
	
	decimalvalue:INT;
	decimalvalueP:INT;
	hexString:STRING(8);
	hexStringP:STRING(8);
	i:INT;
	hexChars:ARRAY [0..15] OF STRING[1]:=['0','1','2','3','4','5','6','7','8','9','A','B','C','D','E','F'];
	index:INT;
END_VAR

(*
 *功能块的作用，把 TxBuffer 缓存区的数据经过 Process Data 的 ComOut 发送出去，
 *而把 ComIn 中的数据接收到 RxBuffer。引用这个功能块的程序执行周期越短，
 *数据交换的效率就越高，所以这段程序应该放在快速任务中作为 Backgroud 代码无条件执行。
*)
IF receive1.Error <> COMERROR_NOERROR THEN
	serialRecError:=TRUE;
END_IF
receive1(
	Prefix:= prefix, 
	Suffix:= suffix, 
	Timeout:=timeout , 
	Reset:= , 
	StringReceived=> , 
	Busy=> , 
	Error=> , 
	RxTimeout=> , 
	ReceivedString:= arr_RcvDataStringTemp, 
	RXbuffer:=gRxBuffer_SRF );

